C01818=1135.613,-74.660,-46.025,178.888,6.133,149.434
C01819=1135.619,-74.910,-46.015,178.885,6.132,149.434
C01820=1135.623,-75.160,-46.005,178.883,6.132,149.434
C01821=1135.629,-75.409,-45.995,178.881,6.131,149.435
C01822=1135.634,-75.659,-45.985,178.879,6.131,149.435
C01823=1135.639,-75.908,-45.975,178.877,6.130,149.436
C01824=1135.645,-76.158,-45.966,178.875,6.130,149.437
C01825=1135.650,-76.409,-45.955,178.872,6.129,149.437
C01826=1135.656,-76.679,-45.944,178.870,6.128,149.438
C01827=1135.662,-76.951,-45.934,178.867,6.128,149.438
C01828=1135.667,-77.223,-45.923,178.866,6.128,149.439
C01829=1135.674,-77.494,-45.912,178.864,6.127,149.439
C01830=1135.678,-77.744,-45.902,178.861,6.127,149.440
C01831=1135.684,-77.994,-45.892,178.859,6.126,149.440
C01832=1135.690,-78.244,-45.883,178.857,6.125,149.441
C01833=1135.695,-78.493,-45.873,178.855,6.125,149.441
C01834=1135.700,-78.743,-45.863,178.853,6.124,149.442
C01835=1135.706,-78.993,-45.853,178.851,6.124,149.442
C01836=1135.710,-79.243,-45.843,178.848,6.123,149.443
C01837=1135.716,-79.492,-45.833,178.846,6.123,149.444
C01838=1135.721,-79.742,-45.824,178.844,6.123,149.444
C01839=1135.727,-79.992,-45.814,178.842,6.122,149.445
C01840=1135.732,-80.241,-45.804,178.840,6.121,149.445
C01841=1135.738,-80.491,-45.795,178.838,6.121,149.446
C01842=1135.743,-80.741,-45.784,178.836,6.121,149.446
C01843=1135.747,-80.991,-45.775,178.833,6.120,149.447
C01844=1135.753,-81.241,-45.765,178.831,6.119,149.447
C01845=1135.759,-81.490,-45.755,178.830,6.119,149.448
C01846=1135.764,-81.739,-45.745,178.827,6.118,149.448
C01847=1135.770,-81.990,-45.736,178.825,6.118,149.449
C01848=1135.775,-82.239,-45.726,178.822,6.117,149.449
C01849=1135.780,-82.490,-45.716,178.821,6.117,149.450
C01850=1135.785,-82.739,-45.706,178.819,6.117,149.450
C01851=1135.790,-82.988,-45.697,178.817,6.116,149.451
C01852=1135.796,-83.239,-45.687,178.815,6.116,149.451
C01853=1135.801,-83.488,-45.677,178.812,6.116,149.452
C01854=1135.807,-83.738,-45.668,178.810,6.115,149.453
C01855=1135.812,-83.987,-45.658,178.808,6.114,149.453
C01856=1135.818,-84.237,-45.649,178.806,6.114,149.453
C01857=1135.822,-84.487,-45.639,178.804,6.113,149.454
C01858=1135.828,-84.738,-45.629,178.802,6.113,149.454
C01859=1135.833,-84.987,-45.620,178.799,6.112,149.455
C01860=1135.839,-85.237,-45.610,178.798,6.112,149.456
C01861=1135.843,-85.486,-45.601,178.795,6.111,149.456
C01862=1135.849,-85.736,-45.591,178.793,6.111,149.457
C01863=1135.854,-85.986,-45.582,178.792,6.111,149.457
C01864=1135.860,-86.236,-45.572,178.789,6.110,149.458
C01865=1135.865,-86.485,-45.562,178.787,6.109,149.458
C01866=1135.871,-86.735,-45.553,178.785,6.109,149.459
C01867=1135.876,-86.984,-45.543,178.783,6.109,149.459
C01868=1135.882,-87.235,-45.534,178.781,6.108,149.460
C01869=1135.886,-87.484,-45.524,178.779,6.107,149.460
C01870=1135.892,-87.735,-45.514,178.777,6.107,149.461
C01871=1135.897,-87.984,-45.505,178.775,6.107,149.461
C01872=1135.903,-88.234,-45.495,178.773,6.106,149.462
C01873=1135.908,-88.484,-45.486,178.771,6.106,149.462
C01874=1135.913,-88.733,-45.477,178.768,6.106,149.463
C01875=1135.919,-88.983,-45.467,178.766,6.105,149.463
C01876=1135.923,-89.232,-45.458,178.764,6.104,149.464
C01877=1135.929,-89.483,-45.448,178.762,6.104,149.464
C01878=1135.934,-89.733,-45.439,178.760,6.103,149.465
C01879=1135.940,-89.982,-45.429,178.758,6.103,149.465
C01880=1135.945,-90.232,-45.420,178.756,6.103,149.466
C01881=1135.950,-90.481,-45.411,178.754,6.102,149.466
C01882=1135.956,-90.731,-45.401,178.751,6.102,149.467
C01883=1135.961,-90.981,-45.392,178.750,6.102,149.467
C01884=1135.967,-91.231,-45.382,178.748,6.101,149.468
C01885=1135.972,-91.481,-45.373,178.745,6.100,149.468
C01886=1135.977,-91.730,-45.364,178.744,6.100,149.469
C01887=1135.983,-91.980,-45.354,178.742,6.099,149.469
C01888=1135.988,-92.230,-45.345,178.739,6.099,149.470
C01889=1135.994,-92.480,-45.336,178.737,6.098,149.471
C01890=1135.999,-92.729,-45.326,178.735,6.098,149.471
C01891=1136.004,-92.979,-45.317,178.733,6.098,149.472
C01892=1136.010,-93.229,-45.308,178.731,6.097,149.472
C01893=1136.015,-93.478,-45.298,178.729,6.097,149.473
C01894=1136.020,-93.728,-45.289,178.727,6.096,149.473
C01895=1136.026,-93.978,-45.280,178.725,6.095,149.474
C01896=1136.031,-94.228,-45.271,178.723,6.096,149.474
C01897=1136.036,-94.478,-45.261,178.721,6.095,149.475
C01898=1136.042,-94.728,-45.252,178.718,6.094,149.475
C01899=1136.047,-94.978,-45.243,178.717,6.094,149.476
C01900=1136.052,-95.227,-45.234,178.715,6.094,149.476
C01901=1136.058,-95.477,-45.224,178.712,6.093,149.477
C01902=1136.063,-95.727,-45.215,178.711,6.093,149.477
C01903=1136.068,-95.977,-45.206,178.709,6.092,149.478
C01904=1136.074,-96.227,-45.196,178.706,6.091,149.478
C01905=1136.079,-96.477,-45.187,178.704,6.092,149.479
C01906=1136.084,-96.725,-45.178,178.702,6.091,149.479
C01907=1136.090,-96.975,-45.169,178.700,6.090,149.480
C01908=1136.095,-97.225,-45.160,178.698,6.090,149.480
C01909=1136.101,-97.475,-45.151,178.696,6.090,149.481
C01910=1136.106,-97.725,-45.142,178.694,6.089,149.481
C01911=1136.111,-97.974,-45.132,178.692,6.089,149.482
C01912=1136.117,-98.224,-45.123,178.690,6.088,149.482
C01913=1136.122,-98.474,-45.114,178.689,6.088,149.483
C01914=1136.127,-98.724,-45.105,178.686,6.087,149.483
C01915=1136.133,-98.974,-45.096,178.684,6.087,149.484
C01916=1136.138,-99.224,-45.087,178.682,6.087,149.484
C01917=1136.143,-99.474,-45.078,178.680,6.086,149.485
C01918=1136.149,-99.722,-45.068,178.678,6.086,149.485
C01919=1136.154,-99.973,-45.059,178.676,6.086,149.486
C01920=1136.160,-100.222,-45.050,178.674,6.085,149.486
C01921=1136.165,-100.472,-45.041,178.672,6.084,149.487
C01922=1136.170,-100.722,-45.032,178.670,6.084,149.487
C01923=1136.175,-100.972,-45.023,178.668,6.083,149.488
C01924=1136.181,-101.222,-45.014,178.666,6.083,149.488
C01925=1136.186,-101.472,-45.005,178.664,6.083,149.489
C01926=1136.191,-101.722,-44.996,178.662,6.082,149.489
C01927=1136.197,-101.971,-44.988,178.660,6.082,149.490
C01928=1136.202,-102.221,-44.979,178.658,6.082,149.490
C01929=1136.208,-102.471,-44.969,178.655,6.081,149.491
C01930=1136.214,-102.743,-44.959,178.654,6.081,149.491
C01931=1136.220,-103.015,-44.949,178.652,6.080,149.492
C01932=1136.225,-103.287,-44.939,178.649,6.080,149.493
C01933=1136.231,-103.560,-44.930,178.647,6.079,149.493
C01934=1136.237,-103.809,-44.921,178.645,6.079,149.494
C01935=1136.242,-104.059,-44.912,178.643,6.078,149.494
C01936=1136.247,-104.309,-44.903,178.641,6.078,149.495
C01937=1136.252,-104.559,-44.894,178.639,6.078,149.495
C01938=1136.258,-104.809,-44.885,178.637,6.077,149.496
C01939=1136.263,-105.059,-44.876,178.635,6.076,149.496
C01940=1136.269,-105.308,-44.868,178.633,6.076,149.497
C01941=1136.274,-105.558,-44.859,178.631,6.075,149.497
C01942=1136.279,-105.807,-44.850,178.629,6.075,149.497
C01943=1136.284,-106.057,-44.841,178.627,6.075,149.498
C01944=1136.290,-106.307,-44.832,178.625,6.074,149.498
C01945=1136.295,-106.557,-44.823,178.623,6.074,149.499
C01946=1136.301,-106.806,-44.815,178.621,6.074,149.500
C01947=1136.306,-107.056,-44.805,178.619,6.074,149.500
C01948=1136.312,-107.306,-44.796,178.617,6.073,149.501
C01949=1136.317,-107.557,-44.788,178.615,6.072,149.501
C01950=1136.322,-107.807,-44.779,178.613,6.072,149.502
C01951=1136.328,-108.056,-44.771,178.611,6.071,149.502
C01952=1136.333,-108.306,-44.762,178.609,6.072,149.503
C01953=1136.338,-108.555,-44.753,178.607,6.071,149.503
C01954=1136.343,-108.805,-44.744,178.605,6.070,149.504
C01955=1136.349,-109.055,-44.735,178.603,6.070,149.504
C01956=1136.354,-109.304,-44.726,178.601,6.069,149.505
C01957=1136.360,-109.554,-44.717,178.600,6.069,149.505
C01958=1136.365,-109.805,-44.709,178.597,6.069,149.505
C01959=1136.370,-110.054,-44.700,178.595,6.068,149.506
C01960=1136.376,-110.304,-44.692,178.594,6.068,149.506
C01961=1136.381,-110.553,-44.683,178.591,6.067,149.507
C01962=1136.386,-110.803,-44.674,178.590,6.067,149.507
C01963=1136.391,-111.053,-44.665,178.588,6.066,149.508
C01964=1136.398,-111.303,-44.657,178.585,6.066,149.508
C01965=1136.403,-111.553,-44.648,178.584,6.066,149.509
C01966=1136.408,-111.803,-44.640,178.582,6.065,149.509
C01967=1136.413,-112.052,-44.631,178.580,6.065,149.510
C01968=1136.419,-112.302,-44.622,178.578,6.064,149.510
C01969=1136.424,-112.551,-44.613,178.576,6.065,149.511
C01970=1136.429,-112.802,-44.605,178.574,6.064,149.512
C01971=1136.435,-113.052,-44.596,178.571,6.063,149.512
C01972=1136.440,-113.301,-44.588,178.570,6.063,149.513
C01973=1136.446,-113.551,-44.579,178.568,6.063,149.513
C01974=1136.451,-113.801,-44.571,178.566,6.063,149.514
C01975=1136.457,-114.050,-44.562,178.564,6.062,149.514
C01976=1136.462,-114.300,-44.553,178.562,6.062,149.514
C01977=1136.467,-114.550,-44.544,178.560,6.061,149.515
C01978=1136.473,-114.801,-44.536,178.558,6.060,149.515
C01979=1136.478,-115.050,-44.528,178.556,6.060,149.516
C01980=1136.484,-115.300,-44.519,178.554,6.060,149.516
C01981=1136.489,-115.549,-44.510,178.552,6.060,149.517
C01982=1136.495,-115.799,-44.502,178.550,6.059,149.517
C01983=1136.500,-116.049,-44.493,178.549,6.059,149.518
C01984=1136.505,-116.299,-44.484,178.546,6.058,149.518
C01985=1136.511,-116.549,-44.476,178.544,6.058,149.519
C01986=1136.516,-116.798,-44.467,178.543,6.058,149.519
C01987=1136.522,-117.048,-44.458,178.540,6.057,149.520
C01988=1136.528,-117.298,-44.451,178.539,6.057,149.520
C01989=1136.532,-117.548,-44.442,178.537,6.056,149.521
C01990=1136.537,-117.798,-44.433,178.535,6.056,149.521
C01991=1136.543,-118.047,-44.426,178.533,6.055,149.522
C01992=1136.548,-118.297,-44.417,178.531,6.056,149.522
C01993=1136.554,-118.547,-44.408,178.529,6.055,149.523
C01994=1136.560,-118.797,-44.400,178.527,6.054,149.523
C01995=1136.565,-119.047,-44.391,178.525,6.054,149.524
C01996=1136.570,-119.297,-44.383,178.523,6.053,149.524
C01997=1136.575,-119.546,-44.375,178.521,6.053,149.525
C01998=1136.581,-119.796,-44.366,178.519,6.053,149.525
C01999=1136.586,-120.046,-44.358,178.518,6.053,149.526
C02000=1136.592,-120.295,-44.349,178.515,6.052,149.526
C02001=1136.597,-120.545,-44.341,178.514,6.052,149.527
C02002=1136.602,-120.796,-44.332,178.512,6.051,149.527
C02003=1136.608,-121.045,-44.324,178.510,6.051,149.528
C02004=1136.613,-121.295,-44.316,178.508,6.051,149.528
C02005=1136.619,-121.544,-44.308,178.506,6.050,149.529
C02006=1136.624,-121.795,-44.300,178.505,6.049,149.529
C02007=1136.629,-122.044,-44.291,178.502,6.049,149.529
C02008=1136.635,-122.294,-44.282,178.501,6.049,149.530
C02009=1136.640,-122.544,-44.274,178.499,6.048,149.530
C02010=1136.645,-122.794,-44.266,178.497,6.048,149.531
C02011=1136.651,-123.043,-44.258,178.495,6.047,149.531
C02012=1136.656,-123.293,-44.249,178.493,6.047,149.532
C02013=1136.662,-123.543,-44.241,178.491,6.047,149.532
C02014=1136.667,-123.793,-44.233,178.489,6.047,149.533
C02015=1136.672,-124.043,-44.225,178.487,6.046,149.533
C02016=1136.678,-124.292,-44.216,178.486,6.046,149.534
C02017=1136.683,-124.543,-44.208,178.483,6.045,149.534
C02018=1136.689,-124.792,-44.199,178.482,6.045,149.535
C02019=1136.694,-125.042,-44.192,178.480,6.045,149.535
C02020=1136.700,-125.291,-44.183,178.478,6.045,149.536
C02021=1136.705,-125.542,-44.175,178.476,6.044,149.536
C02022=1136.710,-125.791,-44.166,178.474,6.043,149.537
C02023=1136.716,-126.041,-44.159,178.472,6.043,149.537
C02024=1136.721,-126.291,-44.151,178.470,6.042,149.538
C02025=1136.727,-126.541,-44.142,178.468,6.042,149.538
C02026=1136.732,-126.791,-44.134,178.466,6.042,149.539
C02027=1136.737,-127.040,-44.126,178.464,6.042,149.539
C02028=1136.743,-127.290,-44.118,178.462,6.041,149.540
C02029=1136.748,-127.540,-44.109,178.461,6.041,149.540
C02030=1136.753,-127.790,-44.102,178.459,6.040,149.540
C02031=1136.759,-128.040,-44.094,178.457,6.040,149.541
C02032=1136.765,-128.289,-44.085,178.455,6.039,149.541
C02033=1136.770,-128.540,-44.077,178.454,6.039,149.542
C02034=1136.349,-128.551,-44.121,178.450,6.043,149.544
C02035=1136.344,-128.300,-44.129,178.452,6.043,149.543
C02036=1136.337,-128.051,-44.137,178.453,6.043,149.543
C02037=1136.333,-127.801,-44.145,178.456,6.044,149.542
C02038=1136.327,-127.551,-44.153,178.457,6.044,149.542
C02039=1136.322,-127.301,-44.162,178.459,6.045,149.541
C02040=1136.316,-127.052,-44.169,178.461,6.045,149.541
C02041=1136.311,-126.802,-44.178,178.463,6.045,149.540
C02042=1136.306,-126.552,-44.186,178.465,6.045,149.540
C02043=1136.300,-126.302,-44.194,178.467,6.046,149.539
C02044=1136.295,-126.052,-44.202,178.469,6.046,149.539
C02045=1136.289,-125.803,-44.210,178.470,6.047,149.539
C02046=1136.284,-125.553,-44.219,178.473,6.048,149.538
C02047=1136.278,-125.303,-44.227,178.474,6.048,149.538
C02048=1136.274,-125.053,-44.235,178.476,6.049,149.537
C02049=1136.268,-124.803,-44.243,178.478,6.049,149.537
C02050=1136.262,-124.554,-44.252,178.480,6.049,149.536
C02051=1136.257,-124.303,-44.260,178.482,6.049,149.536
C02052=1136.252,-124.054,-44.268,178.484,6.050,149.535
C02053=1136.246,-123.804,-44.276,178.486,6.050,149.535
C02054=1136.241,-123.554,-44.285,178.488,6.051,149.534
C02055=1136.235,-123.304,-44.293,178.489,6.051,149.534
C02056=1136.230,-123.055,-44.302,178.492,6.051,149.533
C02057=1136.225,-122.805,-44.309,178.493,6.051,149.533
C02058=1136.219,-122.555,-44.318,178.495,6.052,149.532
C02059=1136.214,-122.305,-44.326,178.497,6.052,149.532
C02060=1136.208,-122.056,-44.335,178.499,6.053,149.531
C02061=1136.203,-121.805,-44.343,178.501,6.053,149.531
C02062=1136.198,-121.556,-44.351,178.503,6.053,149.530
C02063=1136.193,-121.306,-44.360,178.505,6.054,149.530
C02064=1136.187,-121.056,-44.368,178.507,6.054,149.529
C02065=1136.181,-120.807,-44.376,178.509,6.055,149.529
C02066=1136.176,-120.556,-44.385,178.511,6.055,149.528
C02067=1136.171,-120.306,-44.394,178.513,6.056,149.528
C02068=1136.165,-120.057,-44.401,178.514,6.056,149.527
C02069=1136.160,-119.807,-44.410,178.517,6.056,149.527
C02070=1136.155,-119.557,-44.419,178.518,6.056,149.526
C02071=1136.149,-119.308,-44.426,178.520,6.057,149.526
C02072=1136.144,-119.058,-44.435,178.521,6.057,149.526
C02073=1136.138,-118.809,-44.444,178.524,6.058,149.525
C02074=1136.133,-118.558,-44.452,178.526,6.059,149.525
C02075=1136.128,-118.309,-44.460,178.527,6.059,149.524
C02076=1136.122,-118.059,-44.468,178.530,6.060,149.524
C02077=1136.117,-117.809,-44.477,178.531,6.059,149.523
C02078=1136.112,-117.559,-44.486,178.533,6.060,149.523
C02079=1136.106,-117.309,-44.494,178.535,6.060,149.522
C02080=1136.100,-117.059,-44.503,178.537,6.061,149.522
C02081=1136.095,-116.810,-44.512,178.539,6.061,149.521
C02082=1136.089,-116.560,-44.519,178.541,6.062,149.521
C02083=1136.084,-116.310,-44.528,178.543,6.062,149.520
C02084=1136.079,-116.060,-44.537,178.545,6.062,149.520
C02085=1136.074,-115.810,-44.546,178.547,6.063,149.519
C02086=1136.068,-115.561,-44.554,178.549,6.063,149.519
C02087=1136.063,-115.311,-44.562,178.551,6.064,149.518
C02088=1136.058,-115.061,-44.571,178.552,6.064,149.518
C02089=1136.052,-114.811,-44.579,178.555,6.064,149.517
C02090=1136.047,-114.562,-44.588,178.556,6.064,149.517
C02091=1136.042,-114.312,-44.597,178.558,6.065,149.516
C02092=1136.036,-114.063,-44.605,178.561,6.066,149.516
C02093=1136.030,-113.812,-44.613,178.562,6.066,149.515
C02094=1136.025,-113.562,-44.622,178.564,6.067,149.515
C02095=1136.020,-113.312,-44.631,178.566,6.066,149.514
C02096=1136.014,-113.063,-44.640,178.569,6.067,149.514
C02097=1136.009,-112.813,-44.648,178.571,6.068,149.513
C02098=1136.004,-112.563,-44.657,178.572,6.068,149.513
C02099=1135.998,-112.314,-44.665,178.575,6.068,149.512
C02100=1135.993,-112.064,-44.674,178.576,6.068,149.512
C02101=1135.988,-111.814,-44.683,178.578,6.069,149.511
C02102=1135.982,-111.564,-44.691,178.580,6.069,149.511
C02103=1135.976,-111.314,-44.700,178.582,6.070,149.510
C02104=1135.971,-111.065,-44.709,178.584,6.071,149.510
C02105=1135.966,-110.815,-44.718,178.586,6.070,149.509
C02106=1135.961,-110.565,-44.727,178.588,6.071,149.509
C02107=1135.955,-110.315,-44.734,178.590,6.071,149.508
C02108=1135.950,-110.065,-44.743,178.592,6.072,149.508
C02109=1135.944,-109.815,-44.752,178.594,6.073,149.507
C02110=1135.939,-109.566,-44.761,178.596,6.073,149.507
C02111=1135.933,-109.316,-44.770,178.598,6.073,149.506
C02112=1135.928,-109.067,-44.778,178.600,6.073,149.506
C02113=1135.923,-108.817,-44.787,178.602,6.074,149.505
C02114=1135.918,-108.567,-44.796,178.604,6.075,149.505
C02115=1135.912,-108.316,-44.805,178.606,6.075,149.504
C02116=1135.906,-108.067,-44.814,178.608,6.076,149.504
C02117=1135.901,-107.817,-44.822,178.609,6.075,149.503
C02118=1135.896,-107.567,-44.831,178.612,6.076,149.503
C02119=1135.891,-107.317,-44.840,178.614,6.077,149.502
C02120=1135.885,-107.067,-44.849,178.615,6.077,149.502
C02121=1135.880,-106.818,-44.858,178.618,6.078,149.501
C02122=1135.874,-106.568,-44.867,178.619,6.078,149.501
C02123=1135.869,-106.319,-44.875,178.621,6.078,149.500
C02124=1135.864,-106.069,-44.884,178.624,6.079,149.500
C02125=1135.859,-105.819,-44.893,178.626,6.079,149.499
C02126=1135.853,-105.570,-44.902,178.628,6.079,149.499
C02127=1135.847,-105.320,-44.911,178.629,6.079,149.498
C02128=1135.842,-105.070,-44.920,178.632,6.080,149.498
C02129=1135.837,-104.820,-44.929,178.634,6.081,149.497
C02130=1135.832,-104.570,-44.938,178.635,6.081,149.497
C02131=1135.827,-104.320,-44.947,178.638,6.082,149.496
C02132=1135.821,-104.071,-44.955,178.640,6.082,149.496
C02133=1135.816,-103.821,-44.964,178.641,6.082,149.495
C02134=1135.810,-103.571,-44.974,178.644,6.083,149.495
C02135=1135.804,-103.298,-44.983,178.646,6.084,149.494
C02136=1135.798,-103.026,-44.993,178.648,6.083,149.494
C02137=1135.793,-102.754,-45.003,178.650,6.084,149.493
C02138=1135.787,-102.481,-45.013,178.652,6.085,149.493
C02139=1135.781,-102.232,-45.021,178.654,6.085,149.492
C02140=1135.776,-101.982,-45.030,178.656,6.086,149.492
C02141=1135.771,-101.733,-45.039,178.658,6.086,149.491
C02142=1135.765,-101.482,-45.048,178.660,6.086,149.491
C02143=1135.760,-101.233,-45.057,178.663,6.087,149.490
C02144=1135.754,-100.983,-45.066,178.665,6.087,149.490
C02145=1135.750,-100.734,-45.076,178.666,6.087,149.489
C02146=1135.744,-100.484,-45.085,178.669,6.088,149.489
C02147=1135.738,-100.234,-45.094,178.671,6.089,149.488
C02148=1135.733,-99.984,-45.103,178.672,6.089,149.488
C02149=1135.728,-99.735,-45.112,178.674,6.090,149.487
C02150=1135.722,-99.485,-45.121,178.677,6.090,149.487
C02151=1135.717,-99.234,-45.130,178.678,6.090,149.486
C02152=1135.711,-98.985,-45.139,178.680,6.091,149.486
C02153=1135.706,-98.735,-45.148,178.682,6.091,149.485
C02154=1135.701,-98.486,-45.157,178.684,6.092,149.485
C02155=1135.695,-98.235,-45.167,178.687,6.092,149.484
C02156=1135.690,-97.986,-45.176,178.689,6.092,149.484
C02157=1135.685,-97.736,-45.184,178.691,6.093,149.483
C02158=1135.679,-97.487,-45.193,178.693,6.094,149.483
C02159=1135.673,-97.236,-45.203,178.695,6.094,149.482
C02160=1135.669,-96.987,-45.212,178.697,6.094,149.482
C02161=1135.663,-96.737,-45.221,178.699,6.095,149.481
C02162=1135.658,-96.487,-45.230,178.701,6.095,149.481
C02163=1135.652,-96.237,-45.240,178.703,6.096,149.480
C02164=1135.647,-95.987,-45.249,178.705,6.096,149.480
C02165=1135.642,-95.738,-45.258,178.707,6.096,149.479
C02166=1135.636,-95.488,-45.268,178.709,6.097,149.478
C02167=1135.631,-95.238,-45.277,178.711,6.098,149.478
C02168=1135.626,-94.988,-45.285,178.713,6.098,149.477
C02169=1135.621,-94.739,-45.296,178.715,6.098,149.477
C02170=1135.615,-94.489,-45.305,178.717,6.099,149.477
C02171=1135.610,-94.239,-45.313,178.719,6.099,149.476
C02172=1135.604,-93.989,-45.323,178.721,6.100,149.476
C02173=1135.599,-93.740,-45.333,178.723,6.100,149.475
C02174=1135.594,-93.490,-45.341,178.725,6.100,149.474
C02175=1135.588,-93.240,-45.351,178.728,6.101,149.474
C02176=1135.583,-92.990,-45.360,178.730,6.102,149.473
C02177=1135.578,-92.741,-45.369,178.731,6.102,149.473
C02178=1135.572,-92.490,-45.379,178.734,6.102,149.472
C02179=1135.567,-92.241,-45.388,178.736,6.103,149.472
C02180=1135.562,-91.991,-45.398,178.737,6.103,149.471
C02181=1135.556,-91.741,-45.407,178.740,6.104,149.471
C02182=1135.551,-91.491,-45.416,178.742,6.104,149.470
C02183=1135.546,-91.242,-45.426,178.744,6.104,149.470
C02184=1135.541,-90.992,-45.435,178.746,6.105,149.469
C02185=1135.535,-90.742,-45.444,178.748,6.106,149.469
C02186=1135.530,-90.493,-45.454,178.750,6.106,149.468
C02187=1135.525,-90.243,-45.463,178.752,6.106,149.468
C02188=1135.519,-89.993,-45.472,178.754,6.107,149.467
C02189=1135.514,-89.743,-45.482,178.756,6.108,149.467
C02190=1135.508,-89.493,-45.492,178.758,6.107,149.466
C02191=1135.503,-89.244,-45.501,178.761,6.108,149.466
C02192=1135.498,-88.994,-45.510,178.763,6.109,149.465
C02193=1135.492,-88.744,-45.520,178.764,6.109,149.465
C02194=1135.487,-88.495,-45.529,178.767,6.110,149.464
C02195=1135.481,-88.244,-45.539,178.769,6.110,149.464
C02196=1135.476,-87.995,-45.548,178.771,6.111,149.463
C02197=1135.470,-87.745,-45.558,178.773,6.111,149.463
C02198=1135.466,-87.496,-45.567,178.775,6.111,149.462
C02199=1135.460,-87.246,-45.576,178.778,6.112,149.462
C02200=1135.455,-86.996,-45.586,178.779,6.112,149.461
C02201=1135.450,-86.747,-45.595,178.781,6.113,149.461
C02202=1135.444,-86.496,-45.605,178.784,6.114,149.460
C02203=1135.439,-86.247,-45.615,178.785,6.114,149.460
C02204=1135.433,-85.997,-45.624,178.787,6.114,149.459
C02205=1135.429,-85.747,-45.634,178.790,6.115,149.458
C02206=1135.423,-85.497,-45.643,178.792,6.115,149.458
C02207=1135.418,-85.248,-45.653,178.794,6.115,149.457
C02208=1135.412,-84.998,-45.663,178.796,6.116,149.457
C02209=1135.407,-84.748,-45.672,178.798,6.117,149.456
C02210=1135.401,-84.498,-45.682,178.800,6.118,149.456
C02211=1135.396,-84.249,-45.691,178.802,6.117,149.455
C02212=1135.391,-83.999,-45.701,178.805,6.118,149.455
C02213=1135.386,-83.750,-45.710,178.807,6.119,149.454
C02214=1135.380,-83.500,-45.721,178.808,6.119,149.454
C02215=1135.375,-83.249,-45.730,178.811,6.120,149.453
C02216=1135.370,-83.000,-45.740,178.813,6.120,149.453
C02217=1135.364,-82.750,-45.750,178.815,6.121,149.452
C02218=1135.359,-82.501,-45.759,178.817,6.121,149.452
C02219=1135.353,-82.250,-45.769,178.819,6.121,149.451
C02220=1135.348,-82.001,-45.778,178.821,6.122,149.451
C02221=1135.343,-81.752,-45.789,178.824,6.123,149.450
C02222=1135.337,-81.501,-45.798,178.825,6.123,149.450
C02223=1135.333,-81.251,-45.808,178.827,6.124,149.449
C02224=1135.327,-81.001,-45.817,178.830,6.124,149.449
C02225=1135.322,-80.752,-45.827,178.832,6.125,149.448
C02226=1135.316,-80.503,-45.837,178.834,6.125,149.448
C02227=1135.311,-80.253,-45.846,178.836,6.125,149.447
C02228=1135.306,-80.003,-45.856,178.838,6.126,149.447
C02229=1135.301,-79.753,-45.867,178.841,6.127,149.446
C02230=1135.295,-79.503,-45.876,178.843,6.127,149.445
C02231=1135.290,-79.254,-45.886,178.845,6.127,149.445
C02232=1135.284,-79.004,-45.896,178.847,6.128,149.444
C02233=1135.279,-78.754,-45.905,178.849,6.129,149.444
C02234=1135.273,-78.505,-45.915,178.851,6.129,149.444
C02235=1135.268,-78.254,-45.926,178.853,6.129,149.443
C02236=1135.263,-78.004,-45.935,178.856,6.130,149.442
C02237=1135.258,-77.755,-45.945,178.858,6.131,149.442
C02238=1135.252,-77.505,-45.955,178.859,6.131,149.441
C02239=1135.247,-77.233,-45.966,178.862,6.131,149.441
C02240=1135.241,-76.963,-45.976,178.864,6.132,149.440
C02241=1135.235,-76.691,-45.987,178.866,6.133,149.440
C02242=1135.229,-76.419,-45.998,178.869,6.133,149.439
C02243=1135.224,-76.170,-46.008,178.871,6.134,149.438
C02244=1135.218,-75.920,-46.018,178.874,6.134,149.438
C02245=1135.213,-75.670,-46.027,178.875,6.134,149.438
C02246=1135.208,-75.420,-46.038,178.877,6.135,149.437
C02247=1135.202,-75.171,-46.048,178.880,6.136,149.436
C02248=1135.197,-74.921,-46.058,178.882,6.136,149.436
C02249=1135.192,-74.671,-46.067,178.884,6.136,149.435
C02250=1135.187,-74.421,-46.078,178.886,6.137,149.435
C02251=1135.181,-74.171,-46.088,178.888,6.138,149.434
C02252=1135.176,-73.922,-46.097,178.890,6.139,149.434
C02253=1135.171,-73.673,-46.108,178.892,6.138,149.433
C02254=1135.166,-73.422,-46.118,178.895,6.139,149.433
C02255=1135.160,-73.172,-46.128,178.897,6.140,149.432
C02256=1135.154,-72.923,-46.138,178.899,6.140,149.432
C02257=1135.149,-72.673,-46.148,178.901,6.141,149.431
C02258=1135.144,-72.423,-46.158,178.903,6.141,149.431
C02259=1135.139,-72.174,-46.168,178.905,6.142,149.430
C02260=1135.133,-71.924,-46.179,178.908,6.142,149.430
C02261=1135.128,-71.675,-46.188,178.910,6.143,149.429
C02262=1135.123,-71.424,-46.198,178.912,6.144,149.429
C02263=1135.117,-71.175,-46.208,178.914,6.143,149.428
C02264=1135.112,-70.925,-46.218,178.916,6.144,149.427
C02265=1135.106,-70.675,-46.229,178.918,6.145,149.427
C02266=1135.102,-70.426,-46.239,178.921,6.146,149.426
C02267=1135.096,-70.176,-46.249,178.923,6.146,149.426
C02268=1135.091,-69.926,-46.259,178.925,6.146,149.425
C02269=1135.086,-69.676,-46.270,178.927,6.147,149.425
C02270=1135.080,-69.427,-46.280,178.929,6.148,149.424
C02271=1135.074,-69.177,-46.290,178.932,6.148,149.424
C02272=1135.070,-68.927,-46.300,178.934,6.149,149.423
C02273=1135.065,-68.678,-46.310,178.936,6.149,149.423
C02274=1135.059,-68.428,-46.320,178.938,6.149,149.422
C02275=1135.053,-68.179,-46.331,178.940,6.150,149.422
C02276=1135.048,-67.928,-46.341,178.942,6.151,149.421
C02277=1135.043,-67.679,-46.351,178.945,6.151,149.420
C02278=1135.037,-67.429,-46.362,178.947,6.151,149.420
C02279=1135.033,-67.179,-46.372,178.949,6.152,149.420
C02280=1135.027,-66.930,-46.382,178.951,6.153,149.419
C02281=1135.022,-66.680,-46.392,178.953,6.154,149.419
C02282=1135.017,-66.430,-46.403,178.956,6.154,149.418
C02283=1135.011,-66.180,-46.413,178.958,6.155,149.417
C02284=1135.006,-65.930,-46.423,178.960,6.155,149.417
C02285=1135.000,-65.681,-46.434,178.962,6.155,149.416
C02286=1134.995,-65.431,-46.444,178.965,6.156,149.416
C02287=1134.990,-65.181,-46.454,178.967,6.157,149.415
C02288=1134.984,-64.931,-46.465,178.969,6.157,149.415
C02289=1134.979,-64.682,-46.474,178.971,6.158,149.414
C02290=1134.974,-64.432,-46.485,178.973,6.158,149.414
C02291=1134.969,-64.182,-46.495,178.975,6.158,149.413
C02292=1134.963,-63.933,-46.505,178.978,6.159,149.413
C02293=1134.959,-63.683,-46.516,178.980,6.160,149.412
C02294=1134.953,-63.434,-46.527,178.982,6.161,149.412
C02295=1134.948,-63.183,-46.537,178.985,6.161,149.411
C02296=1134.942,-62.934,-46.547,178.986,6.161,149.410
C02297=1134.937,-62.684,-46.558,178.988,6.162,149.410
C02298=1134.932,-62.434,-46.568,178.991,6.163,149.409
C02299=1134.926,-62.184,-46.578,178.993,6.163,149.409
C02300=1134.921,-61.935,-46.590,178.995,6.164,149.408
C02301=1134.916,-61.685,-46.600,178.998,6.165,149.408
C02302=1134.911,-61.435,-46.611,179.000,6.165,149.407
C02303=1134.905,-61.185,-46.621,179.002,6.165,149.407
C02304=1134.900,-60.936,-46.631,179.004,6.166,149.406
C02305=1134.895,-60.686,-46.642,179.006,6.166,149.406
C02306=1134.889,-60.437,-46.652,179.008,6.167,149.405
C02307=1134.884,-60.186,-46.663,179.011,6.168,149.405
C02308=1134.879,-59.937,-46.673,179.013,6.168,149.404
C02309=1134.874,-59.687,-46.684,179.015,6.168,149.404
C02310=1134.869,-59.438,-46.695,179.017,6.169,149.403
C02311=1134.863,-59.188,-46.705,179.019,6.170,149.403
C02312=1134.858,-58.938,-46.716,179.022,6.170,149.402
C02313=1134.852,-58.688,-46.726,179.024,6.171,149.401
C02314=1134.848,-58.439,-46.737,179.026,6.172,149.401
C02315=1134.842,-58.189,-46.747,179.029,6.173,149.400
C02316=1134.837,-57.939,-46.758,179.031,6.173,149.400
C02317=1134.832,-57.690,-46.769,179.033,6.173,149.399
C02318=1134.827,-57.440,-46.779,179.035,6.174,149.399
C02319=1134.821,-57.190,-46.790,179.037,6.174,149.398
C02320=1134.815,-56.940,-46.801,179.040,6.175,149.398
C02321=1134.810,-56.691,-46.812,179.042,6.176,149.397
C02322=1134.805,-56.441,-46.822,179.044,6.176,149.397
C02323=1134.800,-56.191,-46.832,179.046,6.177,149.396
C02324=1134.795,-55.941,-46.844,179.049,6.178,149.395
C02325=1134.789,-55.692,-46.854,179.051,6.178,149.395
C02326=1134.785,-55.442,-46.865,179.053,6.178,149.394
C02327=1134.779,-55.193,-46.875,179.055,6.179,149.394
C02328=1134.774,-54.942,-46.886,179.058,6.179,149.393
C02329=1134.768,-54.693,-46.897,179.060,6.180,149.393
C02330=1134.763,-54.443,-46.908,179.062,6.181,149.392
C02331=1134.757,-54.193,-46.918,179.064,6.182,149.392
C02332=1134.753,-53.944,-46.930,179.067,6.182,149.391
C02333=1134.747,-53.694,-46.940,179.069,6.183,149.391
C02334=1134.742,-53.445,-46.951,179.071,6.183,149.390
C02335=1134.737,-53.194,-46.962,179.073,6.184,149.390
C02336=1134.731,-52.945,-46.973,179.076,6.184,149.389
C02337=1134.726,-52.695,-46.984,179.078,6.185,149.389
C02338=1134.721,-52.445,-46.994,179.080,6.186,149.388
C02339=1134.716,-52.196,-47.005,179.083,6.186,149.387
C02340=1134.710,-51.946,-47.015,179.085,6.187,149.387
C02341=1134.705,-51.696,-47.027,179.087,6.187,149.386
C02342=1134.699,-51.447,-47.038,179.089,6.188,149.386
C02343=1134.694,-51.176,-47.050,179.092,6.189,149.385
C02344=1134.689,-50.905,-47.061,179.094,6.189,149.385
C02345=1134.683,-50.635,-47.073,179.097,6.190,149.384
C02346=1134.677,-50.363,-47.085,179.099,6.191,149.384
C02347=1134.672,-50.114,-47.096,179.101,6.191,149.383
C02348=1134.666,-49.864,-47.106,179.104,6.192,149.382
C02349=1134.661,-49.614,-47.118,179.106,6.192,149.382
C02350=1134.656,-49.365,-47.129,179.108,6.193,149.381
C02351=1134.651,-49.115,-47.140,179.110,6.194,149.381
C02352=1134.645,-48.866,-47.151,179.113,6.194,149.380
C02353=1134.640,-48.615,-47.162,179.115,6.194,149.380
C02354=1134.635,-48.366,-47.173,179.117,6.195,149.379
C02355=1134.629,-48.116,-47.183,179.119,6.196,149.379
C02356=1134.625,-47.867,-47.195,179.122,6.196,149.378
C02357=1134.619,-47.617,-47.206,179.124,6.197,149.378
C02358=1134.614,-47.367,-47.217,179.126,6.198,149.377
C02359=1134.609,-47.118,-47.228,179.129,6.198,149.376
C02360=1134.603,-46.868,-47.239,179.131,6.199,149.376
C02361=1134.598,-46.618,-47.250,179.133,6.200,149.375
C02362=1134.593,-46.368,-47.261,179.135,6.201,149.375
C02363=1134.587,-46.119,-47.272,179.138,6.201,149.374
C02364=1134.582,-45.869,-47.283,179.140,6.202,149.374
C02365=1134.578,-45.619,-47.295,179.142,6.203,149.373
C02366=1134.571,-45.369,-47.306,179.145,6.203,149.373
C02367=1134.567,-45.120,-47.317,179.147,6.204,149.372
C02368=1134.562,-44.870,-47.328,179.149,6.204,149.372
C02369=1134.556,-44.620,-47.339,179.151,6.204,149.371
C02370=1134.551,-44.371,-47.350,179.154,6.205,149.370
C02371=1134.546,-44.121,-47.362,179.156,6.206,149.370
C02372=1134.540,-43.871,-47.372,179.158,6.206,149.370
C02373=1134.535,-43.622,-47.384,179.161,6.207,149.369
C02374=1134.530,-43.372,-47.396,179.163,6.208,149.368
C02375=1134.524,-43.123,-47.406,179.165,6.208,149.368
C02376=1134.519,-42.873,-47.417,179.167,6.209,149.367
C02377=1134.514,-42.623,-47.429,179.170,6.209,149.367
C02378=1134.509,-42.374,-47.440,179.172,6.210,149.366
C02379=1134.503,-42.124,-47.452,179.174,6.211,149.366
C02380=1134.498,-41.874,-47.462,179.177,6.211,149.365
C02381=1134.494,-41.624,-47.474,179.179,6.212,149.365
C02382=1134.488,-41.375,-47.485,179.181,6.213,149.364
C02383=1134.483,-41.125,-47.496,179.184,6.214,149.364
C02384=1134.477,-40.875,-47.508,179.186,6.214,149.363
C02385=1134.472,-40.626,-47.518,179.188,6.215,149.362
C02386=1134.466,-40.376,-47.530,179.191,6.216,149.362
C02387=1134.462,-40.126,-47.542,179.193,6.216,149.361
C02388=1134.456,-39.876,-47.554,179.195,6.217,149.361
C02389=1134.451,-39.627,-47.564,179.198,6.218,149.360
C02390=1134.445,-39.377,-47.576,179.200,6.218,149.360
C02391=1134.441,-39.127,-47.587,179.202,6.219,149.359
C02392=1134.434,-38.878,-47.598,179.205,6.220,149.359
C02393=1134.430,-38.628,-47.610,179.207,6.220,149.358
C02394=1134.424,-38.378,-47.622,179.210,6.221,149.357
C02395=1134.420,-38.129,-47.633,179.212,6.222,149.357
C02396=1134.414,-37.879,-47.645,179.214,6.222,149.357
C02397=1134.409,-37.630,-47.656,179.217,6.223,149.356
C02398=1134.404,-37.380,-47.668,179.219,6.224,149.355
C02399=1134.399,-37.129,-47.678,179.221,6.224,149.355
C02400=1134.393,-36.880,-47.690,179.223,6.225,149.354
C02401=1134.388,-36.631,-47.701,179.226,6.225,149.354
C02402=1134.382,-36.381,-47.713,179.228,6.226,149.353
C02403=1134.378,-36.131,-47.724,179.230,6.227,149.353
C02404=1134.372,-35.881,-47.736,179.233,6.227,149.352
C02405=1134.368,-35.631,-47.747,179.235,6.228,149.352
C02406=1134.362,-35.382,-47.759,179.237,6.229,149.351
C02407=1134.356,-35.132,-47.771,179.239,6.230,149.351
C02408=1134.351,-34.883,-47.782,179.242,6.230,149.350
C02409=1134.346,-34.633,-47.794,179.244,6.231,149.349
C02410=1134.341,-34.383,-47.805,179.246,6.232,149.349
C02411=1134.335,-34.134,-47.817,179.249,6.232,149.348
C02412=1134.330,-33.884,-47.829,179.251,6.233,149.348
C02413=1134.325,-33.634,-47.840,179.253,6.234,149.347
C02414=1134.320,-33.384,-47.852,179.256,6.234,149.347
C02415=1134.315,-33.135,-47.863,179.258,6.235,149.346
C02416=1134.310,-32.885,-47.875,179.260,6.236,149.346
C02417=1134.304,-32.636,-47.886,179.263,6.236,149.345
C02418=1134.299,-32.386,-47.898,179.265,6.237,149.344
C02419=1134.293,-32.136,-47.910,179.268,6.238,149.344
C02420=1134.288,-31.887,-47.922,179.270,6.238,149.344
C02421=1134.284,-31.637,-47.934,179.272,6.239,149.343
C02422=1134.278,-31.387,-47.945,179.275,6.240,149.342
C02423=1134.273,-31.138,-47.957,179.277,6.240,149.342
C02424=1134.267,-30.888,-47.968,179.279,6.241,149.341
C02425=1134.262,-30.638,-47.980,179.282,6.242,149.341
C02426=1134.257,-30.389,-47.991,179.284,6.242,149.340
C02427=1134.252,-30.139,-48.003,179.286,6.243,149.340
C02428=1134.247,-29.889,-48.016,179.289,6.243,149.339
C02429=1134.241,-29.640,-48.028,179.291,6.244,149.339
C02430=1134.237,-29.390,-48.039,179.293,6.245,149.338
C02431=1134.231,-29.140,-48.051,179.296,6.245,149.337
C02432=1134.226,-28.890,-48.063,179.298,6.246,149.337
C02433=1134.221,-28.641,-48.074,179.300,6.247,149.336
C02434=1134.215,-28.392,-48.086,179.303,6.248,149.336
C02435=1134.210,-28.142,-48.098,179.305,6.249,149.335
C02436=1134.205,-27.892,-48.110,179.308,6.250,149.335
C02437=1134.200,-27.642,-48.121,179.310,6.250,149.334
C02438=1134.195,-27.393,-48.134,179.313,6.251,149.334
C02439=1134.189,-27.143,-48.146,179.315,6.252,149.333
C02440=1134.184,-26.893,-48.158,179.317,6.252,149.332
C02441=1134.179,-26.643,-48.169,179.320,6.253,149.332
C02442=1134.174,-26.394,-48.182,179.322,6.254,149.332
C02443=1134.169,-26.144,-48.194,179.324,6.254,149.331
C02444=1134.163,-25.894,-48.205,179.327,6.255,149.330
C02445=1134.158,-25.645,-48.217,179.329,6.256,149.330
C02446=1134.153,-25.395,-48.229,179.331,6.256,149.329
C02447=1134.147,-25.126,-48.242,179.334,6.258,149.329
C02448=1134.142,-24.855,-48.255,179.337,6.258,149.328
C02449=1134.136,-24.585,-48.268,179.339,6.259,149.328
C02450=1134.130,-24.315,-48.281,179.342,6.259,149.327
C02451=1134.125,-24.065,-48.293,179.344,6.260,149.326
C02452=1134.120,-23.816,-48.305,179.346,6.261,149.326
C02453=1134.115,-23.566,-48.317,179.348,6.262,149.325
C02454=1134.110,-23.316,-48.329,179.352,6.263,149.325
C02455=1134.104,-23.067,-48.341,179.354,6.264,149.324
C02456=1134.099,-22.817,-48.353,179.356,6.264,149.324
C02457=1134.094,-22.567,-48.365,179.359,6.265,149.323
C02458=1134.088,-22.318,-48.378,179.361,6.266,149.323
C02459=1134.084,-22.068,-48.389,179.363,6.266,149.322
C02460=1134.079,-21.819,-48.402,179.366,6.267,149.321
C02461=1134.073,-21.569,-48.413,179.368,6.268,149.321
C02462=1134.068,-21.320,-48.426,179.370,6.268,149.321
C02463=1134.063,-21.070,-48.438,179.373,6.269,149.320
C02464=1134.057,-20.820,-48.450,179.375,6.270,149.319
C02465=1134.052,-20.570,-48.462,179.378,6.271,149.319
C02466=1134.047,-20.320,-48.474,179.380,6.271,149.318
C02467=1134.042,-20.071,-48.487,179.382,6.272,149.318
C02468=1134.036,-19.821,-48.499,179.385,6.273,149.317
C02469=1134.031,-19.572,-48.511,179.387,6.273,149.317
C02470=1134.026,-19.322,-48.523,179.389,6.274,149.316
C02471=1134.021,-19.073,-48.535,179.392,6.275,149.316
C02472=1134.016,-18.822,-48.548,179.394,6.275,149.315
C02473=1134.011,-18.573,-48.560,179.397,6.276,149.314
C02474=1134.006,-18.323,-48.572,179.399,6.278,149.314
C02475=1134.001,-18.074,-48.585,179.402,6.278,149.313
C02476=1133.995,-17.824,-48.597,179.404,6.279,149.313
C02477=1133.990,-17.574,-48.609,179.406,6.280,149.312
C02478=1133.985,-17.324,-48.621,179.409,6.281,149.312
C02479=1133.980,-17.075,-48.634,179.411,6.281,149.311
C02480=1133.974,-16.826,-48.646,179.413,6.282,149.311
C02481=1133.969,-16.576,-48.658,179.416,6.283,149.310
C02482=1133.964,-16.327,-48.671,179.419,6.284,149.310
C02483=1133.958,-16.077,-48.683,179.421,6.285,149.309
C02484=1133.954,-15.827,-48.696,179.423,6.285,149.309
C02485=1133.949,-15.577,-48.708,179.426,6.286,149.308
C02486=1133.943,-15.327,-48.720,179.428,6.287,149.307
C02487=1133.938,-15.078,-48.733,179.430,6.287,149.307
C02488=1133.933,-14.829,-48.745,179.433,6.288,149.306
C02489=1133.928,-14.579,-48.757,179.435,6.289,149.306
C02490=1133.923,-14.329,-48.770,179.438,6.290,149.305
C02491=1133.917,-14.080,-48.783,179.440,6.291,149.305
C02492=1133.912,-13.829,-48.795,179.443,6.291,149.304
C02493=1133.907,-13.580,-48.808,179.445,6.292,149.304
C02494=1133.902,-13.331,-48.820,179.447,6.293,149.303
C02495=1133.896,-13.081,-48.832,179.450,6.293,149.303
C02496=1133.891,-12.831,-48.845,179.452,6.295,149.302
C02497=1133.886,-12.582,-48.857,179.455,6.295,149.301
C02498=1133.880,-12.332,-48.869,179.457,6.296,149.301
C02499=1133.876,-12.082,-48.882,179.459,6.297,149.300
C02500=1133.871,-11.833,-48.895,179.462,6.297,149.300
C02501=1133.866,-11.583,-48.908,179.464,6.298,149.299
C02502=1133.860,-11.333,-48.920,179.467,6.299,149.299
C02503=1133.854,-11.084,-48.933,179.470,6.300,149.298
C02504=1133.850,-10.834,-48.946,179.472,6.301,149.298
C02505=1133.845,-10.585,-48.958,179.474,6.302,149.297
C02506=1133.840,-10.335,-48.971,179.477,6.302,149.296
C02507=1133.834,-10.085,-48.983,179.479,6.303,149.296
C02508=1133.829,-9.836,-48.995,179.481,6.304,149.296
C02509=1133.825,-9.586,-49.008,179.484,6.305,149.295
C02510=1133.819,-9.336,-49.021,179.487,6.306,149.294
C02511=1133.814,-9.087,-49.034,179.489,6.307,149.294
C02512=1133.808,-8.838,-49.047,179.491,6.307,149.293
C02513=1133.804,-8.587,-49.059,179.494,6.308,149.293
C02514=1133.799,-8.338,-49.071,179.496,6.309,149.292
C02515=1133.793,-8.088,-49.085,179.499,6.310,149.292
C02516=1133.788,-7.839,-49.097,179.501,6.311,149.291
C02517=1133.782,-7.589,-49.110,179.503,6.311,149.291
C02518=1133.778,-7.339,-49.123,179.506,6.312,149.290
C02519=1133.773,-7.090,-49.135,179.508,6.313,149.289
C02520=1133.767,-6.840,-49.149,179.511,6.314,149.289
C02521=1133.762,-6.591,-49.161,179.514,6.315,149.288
C02522=1133.757,-6.341,-49.174,179.516,6.315,149.288
C02523=1133.752,-6.091,-49.186,179.518,6.316,149.287
C02524=1133.746,-5.842,-49.199,179.521,6.317,149.287
C02525=1133.741,-5.592,-49.212,179.523,6.318,149.286
C02526=1133.736,-5.342,-49.225,179.526,6.319,149.286
C02527=1133.731,-5.093,-49.237,179.528,6.319,149.285
C02528=1133.725,-4.843,-49.251,179.531,6.320,149.285
C02529=1133.721,-4.593,-49.264,179.533,6.321,149.284
C02530=1133.716,-4.344,-49.276,179.536,6.322,149.283
C02531=1133.710,-4.094,-49.289,179.538,6.323,149.283
C02532=1133.705,-3.844,-49.302,179.540,6.324,149.282
C02533=1133.700,-3.595,-49.315,179.543,6.324,149.282
C02534=1133.694,-3.345,-49.328,179.545,6.325,149.281
C02535=1133.690,-3.095,-49.341,179.548,6.327,149.281
C02536=1133.685,-2.846,-49.354,179.551,6.327,149.280
C02537=1133.679,-2.597,-49.368,179.553,6.328,149.280
C02538=1133.674,-2.348,-49.380,179.555,6.329,149.279
C02539=1133.669,-2.098,-49.393,179.558,6.330,149.279
C02540=1133.664,-1.848,-49.406,179.560,6.331,149.278
C02541=1133.658,-1.599,-49.419,179.563,6.331,149.278
C02542=1133.654,-1.349,-49.432,179.565,6.332,149.277
C02543=1133.648,-1.099,-49.445,179.567,6.333,149.276
C02544=1133.643,-0.850,-49.458,179.570,6.334,149.276
C02545=1133.638,-0.600,-49.471,179.573,6.335,149.275
C02546=1133.633,-0.350,-49.484,179.575,6.335,149.275
C02547=1133.628,-0.101,-49.498,179.577,6.336,149.274
C02548=1133.623,0.149,-49.511,179.580,6.337,149.274
C02549=1133.617,0.398,-49.523,179.583,6.338,149.273
C02550=1133.612,0.649,-49.537,179.585,6.339,149.273
C02551=1133.607,0.918,-49.550,179.588,6.340,149.272
C02552=1133.601,1.187,-49.565,179.590,6.341,149.272
C02553=1133.596,1.457,-49.579,179.593,6.341,149.271
C02554=1133.590,1.726,-49.593,179.596,6.343,149.270
C02555=1133.585,1.976,-49.607,179.598,6.343,149.270
C02556=1133.580,2.225,-49.620,179.600,6.344,149.269
C02557=1133.575,2.475,-49.633,179.603,6.346,149.269
C02558=1133.569,2.725,-49.646,179.606,6.346,149.268
C02559=1133.564,2.973,-49.659,179.608,6.347,149.268
C02560=1133.559,3.224,-49.673,179.610,6.348,149.267
C02561=1133.554,3.473,-49.685,179.614,6.349,149.267
C02562=1133.549,3.723,-49.699,179.616,6.350,149.266
C02563=1133.544,3.972,-49.712,179.618,6.351,149.266
C02564=1133.539,4.222,-49.726,179.621,6.351,149.265
C02565=1133.534,4.472,-49.738,179.623,6.353,149.264
C02566=1133.529,4.721,-49.753,179.626,6.354,149.264
C02567=1133.524,4.971,-49.765,179.628,6.354,149.263
C02568=1133.518,5.220,-49.779,179.630,6.355,149.263
C02569=1133.513,5.470,-49.792,179.633,6.356,149.262
C02570=1133.508,5.719,-49.805,179.636,6.357,149.262
C02571=1133.503,5.969,-49.818,179.638,6.358,149.261
C02572=1133.498,6.218,-49.832,179.641,6.359,149.261
C02573=1133.492,6.469,-49.846,179.643,6.360,149.260
C02574=1133.487,6.717,-49.859,179.646,6.360,149.260
C02575=1133.482,6.968,-49.873,179.648,6.361,149.259
C02576=1133.477,7.217,-49.885,179.651,6.362,149.258
C02577=1133.472,7.467,-49.900,179.653,6.363,149.258
C02578=1133.467,7.716,-49.912,179.655,6.364,149.258
C02579=1133.462,7.966,-49.926,179.659,6.365,149.257
C02580=1133.456,8.216,-49.940,179.661,6.366,149.256
C02581=1133.452,8.466,-49.953,179.663,6.367,149.256
C02582=1133.446,8.715,-49.967,179.666,6.367,149.255
C02583=1133.441,8.965,-49.980,179.668,6.369,149.255
C02584=1133.436,9.214,-49.993,179.671,6.370,149.254
C02585=1133.431,9.464,-50.007,179.673,6.370,149.254
C02586=1133.426,9.713,-50.020,179.676,6.372,149.253
C02587=1133.421,9.963,-50.034,179.678,6.373,149.253
C02588=1133.415,10.212,-50.048,179.681,6.373,149.252
C02589=1133.411,10.462,-50.061,179.684,6.375,149.252
C02590=1133.405,10.711,-50.075,179.686,6.375,149.251
C02591=1133.400,10.961,-50.088,179.688,6.376,149.250
C02592=1133.396,11.211,-50.102,179.691,6.377,149.250
C02593=1133.390,11.460,-50.116,179.693,6.378,149.249
C02594=1133.385,11.710,-50.129,179.696,6.379,149.249
C02595=1133.380,11.959,-50.143,179.698,6.379,149.248
C02596=1133.375,12.209,-50.156,179.701,6.381,149.248
C02597=1133.369,12.458,-50.170,179.704,6.382,149.247
C02598=1133.364,12.708,-50.184,179.706,6.382,149.247
C02599=1133.360,12.958,-50.197,179.709,6.384,149.246
C02600=1133.354,13.207,-50.211,179.711,6.384,149.246
C02601=1133.349,13.457,-50.225,179.713,6.385,149.245
C02602=1133.343,13.706,-50.239,179.716,6.387,149.245
C02603=1133.339,13.956,-50.252,179.719,6.387,149.244
C02604=1133.333,14.205,-50.266,179.721,6.388,149.244
C02605=1133.328,14.455,-50.280,179.724,6.390,149.243
C02606=1133.323,14.705,-50.294,179.726,6.390,149.242
C02607=1133.318,14.954,-50.307,179.729,6.391,149.242
C02608=1133.313,15.204,-50.321,179.731,6.392,149.241
C02609=1133.308,15.453,-50.335,179.734,6.393,149.241
C02610=1133.302,15.703,-50.349,179.736,6.394,149.240
C02611=1133.298,15.952,-50.362,179.739,6.395,149.240
C02612=1133.293,16.201,-50.376,179.742,6.396,149.239
C02613=1133.288,16.451,-50.390,179.744,6.397,149.239
C02614=1133.282,16.701,-50.404,179.747,6.398,149.238
C02615=1133.277,16.950,-50.418,179.749,6.399,149.238
C02616=1133.272,17.200,-50.432,179.752,6.400,149.237
C02617=1133.268,17.450,-50.446,179.754,6.401,149.237
C02618=1133.262,17.699,-50.459,179.757,6.401,149.236
C02619=1133.257,17.949,-50.473,179.760,6.403,149.235
C02620=1133.252,18.199,-50.488,179.762,6.404,149.235
C02621=1133.246,18.448,-50.502,179.764,6.404,149.234
C02622=1133.241,18.697,-50.516,179.767,6.406,149.234
C02623=1133.236,18.948,-50.529,179.769,6.407,149.233
C02624=1133.231,19.196,-50.543,179.772,6.408,149.233
C02625=1133.226,19.446,-50.557,179.775,6.409,149.232
C02626=1133.221,19.696,-50.571,179.777,6.410,149.232
C02627=1133.216,19.945,-50.586,179.780,6.411,149.231
C02628=1133.211,20.194,-50.599,179.782,6.412,149.231
C02629=1133.206,20.444,-50.614,179.785,6.412,149.230
C02630=1133.201,20.695,-50.627,179.787,6.414,149.230
C02631=1133.195,20.944,-50.641,179.790,6.414,149.229
C02632=1133.190,21.193,-50.655,179.792,6.415,149.229
C02633=1133.185,21.443,-50.670,179.795,6.417,149.228
C02634=1133.180,21.693,-50.684,179.798,6.417,149.228
C02635=1133.175,21.942,-50.698,179.800,6.419,149.227
C02636=1133.170,22.191,-50.712,179.802,6.420,149.227
C02637=1133.166,22.441,-50.726,179.805,6.420,149.226
C02638=1133.161,22.690,-50.740,179.808,6.422,149.225
C02639=1133.155,22.939,-50.754,179.810,6.423,149.225
C02640=1133.150,23.189,-50.768,179.813,6.424,149.224
C02641=1133.145,23.439,-50.783,179.816,6.425,149.224
C02642=1133.140,23.689,-50.797,179.818,6.425,149.223
C02643=1133.135,23.938,-50.811,179.821,6.427,149.223
C02644=1133.130,24.187,-50.825,179.823,6.428,149.222
C02645=1133.125,24.437,-50.839,179.826,6.429,149.222
C02646=1133.120,24.687,-50.854,179.829,6.430,149.221
C02647=1133.115,24.936,-50.868,179.831,6.430,149.221
C02648=1133.109,25.185,-50.882,179.833,6.432,149.220
C02649=1133.104,25.436,-50.897,179.836,6.432,149.220
C02650=1133.099,25.685,-50.911,179.839,6.434,149.219
C02651=1133.094,25.935,-50.925,179.841,6.435,149.219
C02652=1133.089,26.185,-50.940,179.844,6.435,149.218
C02653=1133.083,26.433,-50.954,179.846,6.437,149.217
C02654=1133.078,26.683,-50.968,179.849,6.438,149.217
C02655=1133.073,26.952,-50.983,179.852,6.439,149.216
C02656=1133.068,27.221,-50.999,179.855,6.441,149.216
C02657=1133.062,27.490,-51.014,179.857,6.441,149.215
C02658=1133.057,27.759,-51.030,179.860,6.443,149.215
C02659=1133.051,28.008,-51.044,179.862,6.443,149.214
C02660=1133.046,28.258,-51.059,179.865,6.445,149.214
C02661=1133.041,28.507,-51.074,179.868,6.446,149.213
C02662=1133.036,28.757,-51.088,179.870,6.446,149.213
C02663=1133.032,29.007,-51.102,179.873,6.448,149.212
C02664=1133.027,29.256,-51.116,179.875,6.448,149.212
C02665=1133.021,29.506,-51.131,179.878,6.450,149.211
C02666=1133.016,29.755,-51.146,179.881,6.450,149.210
C02667=1133.011,30.005,-51.160,179.883,6.452,149.210
C02668=1133.006,30.254,-51.174,179.886,6.453,149.210
C02669=1133.001,30.504,-51.189,179.889,6.454,149.209
C02670=1132.996,30.753,-51.204,179.891,6.455,149.208
C02671=1132.990,31.003,-51.219,179.894,6.457,149.208
C02672=1132.985,31.253,-51.233,179.896,6.457,149.207
C02673=1132.981,31.502,-51.247,179.899,6.458,149.207
C02674=1132.976,31.752,-51.262,179.901,6.459,149.206
C02675=1132.971,32.001,-51.276,179.904,6.460,149.206
C02676=1132.965,32.251,-51.291,179.907,6.461,149.205
C02677=1132.960,32.500,-51.306,179.909,6.462,149.205
C02678=1132.955,32.749,-51.320,179.912,6.464,149.204
C02679=1132.950,32.999,-51.335,179.914,6.464,149.204
C02680=1132.945,33.249,-51.350,179.917,6.466,149.203
C02681=1132.940,33.498,-51.364,179.919,6.467,149.203
C02682=1132.935,33.748,-51.379,179.923,6.468,149.202
C02683=1132.930,33.997,-51.394,179.925,6.469,149.202
C02684=1132.924,34.247,-51.409,179.927,6.470,149.201
C02685=1132.920,34.496,-51.424,179.930,6.471,149.200
C02686=1132.915,34.746,-51.438,179.932,6.472,149.200
C02687=1132.910,34.996,-51.452,179.935,6.473,149.200
C02688=1132.904,35.245,-51.468,179.937,6.474,149.199
C02689=1132.900,35.495,-51.482,179.940,6.475,149.198
C02690=1132.895,35.744,-51.497,179.943,6.476,149.198
C02691=1132.889,35.994,-51.512,179.945,6.478,149.198
C02692=1132.885,36.243,-51.527,179.948,6.478,149.197
C02693=1132.880,36.493,-51.541,179.951,6.480,149.196
C02694=1132.874,36.742,-51.557,179.953,6.481,149.196
C02695=1132.869,36.992,-51.571,179.956,6.482,149.195
C02696=1132.865,37.241,-51.586,179.958,6.483,149.195
C02697=1132.859,37.491,-51.601,179.961,6.484,149.194
C02698=1132.854,37.740,-51.616,179.964,6.485,149.194
C02699=1132.849,37.990,-51.631,179.967,6.487,149.193
C02700=1132.844,38.239,-51.646,179.969,6.487,149.193
C02701=1132.839,38.489,-51.660,179.971,6.489,149.192
C02702=1132.834,38.738,-51.676,179.974,6.489,149.192
C02703=1132.829,38.987,-51.691,179.977,6.491,149.191
C02704=1132.823,39.237,-51.705,179.979,6.492,149.191
C02705=1132.819,39.486,-51.720,179.982,6.493,149.190
C02706=1132.814,39.736,-51.735,179.984,6.494,149.190
C02707=1132.808,39.985,-51.750,179.987,6.496,149.189
C02708=1132.804,40.235,-51.765,179.990,6.496,149.189
C02709=1132.798,40.485,-51.780,179.993,6.498,149.188
C02710=1132.793,40.734,-51.795,179.995,6.499,149.188
C02711=1132.788,40.983,-51.811,179.998,6.500,149.187
C02712=1132.783,41.233,-51.825,-179.999,6.501,149.187
C02713=1132.778,41.482,-51.841,-179.997,6.502,149.186
C02714=1132.773,41.731,-51.856,-179.994,6.504,149.186
C02715=1132.767,41.981,-51.870,-179.992,6.504,149.185
C02716=1132.763,42.231,-51.886,-179.989,6.506,149.185
C02717=1132.758,42.480,-51.901,-179.987,6.507,149.184
C02718=1132.753,42.730,-51.916,-179.984,6.508,149.184
C02719=1132.747,42.980,-51.931,-179.981,6.509,149.183
C02720=1132.743,43.229,-51.946,-179.979,6.510,149.183
C02721=1132.737,43.478,-51.962,-179.976,6.511,149.182
C02722=1132.732,43.728,-51.976,-179.973,6.512,149.181
C02723=1132.727,43.977,-51.992,-179.970,6.514,149.181
C02724=1132.722,44.226,-52.007,-179.968,6.515,149.180
C02725=1132.718,44.476,-52.023,-179.965,6.516,149.180
C02726=1132.713,44.726,-52.037,-179.963,6.517,149.179
C02727=1132.707,44.975,-52.052,-179.960,6.519,149.179
C02728=1132.703,45.225,-52.067,-179.958,6.519,149.178
C02729=1132.697,45.474,-52.083,-179.955,6.521,149.178
C02730=1132.692,45.723,-52.099,-179.952,6.522,149.177
C02731=1132.687,45.972,-52.114,-179.950,6.523,149.177
C02732=1132.682,46.223,-52.129,-179.946,6.524,149.176
C02733=1132.677,46.472,-52.144,-179.944,6.525,149.176
C02734=1132.672,46.722,-52.159,-179.942,6.527,149.175
C02735=1132.667,46.971,-52.175,-179.939,6.528,149.175
C02736=1132.662,47.220,-52.190,-179.936,6.529,149.174
C02737=1132.657,47.470,-52.206,-179.934,6.530,149.174
C02738=1132.653,47.719,-52.221,-179.931,6.531,149.173
C02739=1132.647,47.969,-52.237,-179.929,6.532,149.173
C02740=1132.642,48.218,-52.252,-179.926,6.533,149.172
C02741=1132.637,48.467,-52.267,-179.923,6.535,149.172
C02742=1132.632,48.717,-52.283,-179.921,6.536,149.171
C02743=1132.627,48.967,-52.299,-179.918,6.537,149.171
C02744=1132.622,49.216,-52.314,-179.915,6.538,149.170
C02745=1132.617,49.465,-52.329,-179.913,6.540,149.170
C02746=1132.612,49.715,-52.345,-179.910,6.541,149.169
C02747=1132.607,49.964,-52.360,-179.907,6.542,149.169
C02748=1132.602,50.214,-52.376,-179.905,6.543,149.168
C02749=1132.597,50.463,-52.391,-179.902,6.544,149.168
C02750=1132.592,50.712,-52.406,-179.899,6.545,149.167
C02751=1132.587,50.962,-52.422,-179.896,6.547,149.167
C02752=1132.582,51.212,-52.438,-179.894,6.548,149.166
C02753=1132.577,51.461,-52.454,-179.891,6.550,149.166
C02754=1132.572,51.711,-52.469,-179.889,6.550,149.165
C02755=1132.567,51.960,-52.484,-179.886,6.552,149.165
C02756=1132.562,52.210,-52.500,-179.883,6.553,149.164
C02757=1132.556,52.459,-52.516,-179.881,6.554,149.164
C02758=1132.552,52.709,-52.531,-179.878,6.555,149.163
C02759=1132.547,52.978,-52.548,-179.875,6.557,149.163
C02760=1132.541,53.246,-52.565,-179.872,6.557,149.162
C02761=1132.536,53.515,-52.582,-179.870,6.559,149.162
C02762=1132.530,53.783,-52.599,-179.866,6.560,149.161
C02763=1132.525,54.033,-52.615,-179.864,6.562,149.160
C02764=1132.520,54.283,-52.631,-179.862,6.563,149.160
C02765=1132.515,54.532,-52.646,-179.859,6.564,149.160
C02766=1132.510,54.781,-52.661,-179.856,6.566,149.159
C02767=1132.505,55.030,-52.678,-179.853,6.567,149.158
C02768=1132.500,55.280,-52.693,-179.851,6.568,149.158
C02769=1132.495,55.529,-52.709,-179.848,6.569,149.158
C02770=1132.490,55.779,-52.725,-179.845,6.570,149.157
C02771=1132.485,56.028,-52.740,-179.842,6.572,149.156
C02772=1132.480,56.277,-52.756,-179.840,6.573,149.156
C02773=1132.475,56.527,-52.772,-179.838,6.574,149.156
C02774=1132.470,56.777,-52.788,-179.834,6.576,149.155
C02775=1132.465,57.027,-52.804,-179.832,6.576,149.154
C02776=1132.460,57.276,-52.820,-179.829,6.578,149.154
C02777=1132.455,57.525,-52.836,-179.827,6.580,149.154
C02778=1132.450,57.775,-52.852,-179.824,6.580,149.153
C02779=1132.445,58.024,-52.868,-179.821,6.582,149.152
C02780=1132.439,58.273,-52.884,-179.819,6.583,149.152
C02781=1132.435,58.523,-52.899,-179.816,6.584,149.152
C02782=1132.430,58.772,-52.915,-179.813,6.586,149.151
C02783=1132.425,59.022,-52.931,-179.811,6.586,149.150
C02784=1132.420,59.271,-52.947,-179.808,6.588,149.150
C02785=1132.415,59.520,-52.963,-179.805,6.590,149.150
C02786=1132.410,59.770,-52.979,-179.803,6.590,149.149
C02787=1132.405,60.019,-52.995,-179.800,6.592,149.149
C02788=1132.400,60.269,-53.011,-179.797,6.593,149.148
C02789=1132.395,60.518,-53.028,-179.795,6.594,149.148
C02790=1132.390,60.767,-53.043,-179.792,6.596,149.147
C02791=1132.385,61.017,-53.059,-179.789,6.597,149.147
C02792=1132.380,61.266,-53.075,-179.787,6.598,149.146
C02793=1132.375,61.516,-53.091,-179.784,6.600,149.146
C02794=1132.370,61.765,-53.108,-179.781,6.601,149.145
C02795=1132.365,62.015,-53.124,-179.778,6.603,149.145
C02796=1132.360,62.264,-53.140,-179.776,6.603,149.144
C02797=1132.355,62.514,-53.156,-179.773,6.605,149.144
C02798=1132.350,62.763,-53.172,-179.770,6.606,149.143
C02799=1132.346,63.013,-53.188,-179.768,6.607,149.143
C02800=1132.341,63.262,-53.204,-179.765,6.609,149.142
C02801=1132.335,63.512,-53.221,-179.762,6.610,149.142
C02802=1132.330,63.761,-53.237,-179.760,6.611,149.141
C02803=1132.325,64.010,-53.254,-179.757,6.613,149.141
C02804=1132.320,64.260,-53.270,-179.754,6.614,149.140
C02805=1132.316,64.509,-53.286,-179.752,6.615,149.140
C02806=1132.310,64.759,-53.302,-179.749,6.616,149.139
C02807=1132.306,65.008,-53.318,-179.746,6.618,149.139
C02808=1132.301,65.257,-53.335,-179.743,6.620,149.138
C02809=1132.296,65.507,-53.351,-179.741,6.620,149.138
C02810=1132.291,65.756,-53.367,-179.738,6.622,149.137
C02811=1132.285,66.006,-53.384,-179.735,6.623,149.137
C02812=1132.280,66.255,-53.400,-179.733,6.624,149.136
C02813=1132.276,66.505,-53.417,-179.730,6.626,149.136
C02814=1132.270,66.754,-53.432,-179.728,6.627,149.135
C02815=1132.266,67.004,-53.449,-179.724,6.629,149.135
C02816=1132.261,67.252,-53.465,-179.722,6.630,149.134
C02817=1132.256,67.502,-53.482,-179.719,6.631,149.134
C02818=1132.251,67.752,-53.498,-179.717,6.633,149.133
C02819=1132.246,68.001,-53.515,-179.714,6.633,149.133
C02820=1132.241,68.250,-53.531,-179.711,6.635,149.132
C02821=1132.236,68.500,-53.547,-179.709,6.637,149.132
C02822=1132.231,68.750,-53.564,-179.706,6.638,149.131
C02823=1132.225,68.998,-53.580,-179.704,6.639,149.131
C02824=1132.221,69.248,-53.597,-179.700,6.640,149.130
C02825=1132.217,69.497,-53.614,-179.698,6.642,149.130
C02826=1132.210,69.747,-53.630,-179.695,6.644,149.129
C02827=1132.206,69.997,-53.647,-179.693,6.644,149.129
C02828=1132.201,70.245,-53.663,-179.690,6.646,149.128
C02829=1132.196,70.495,-53.680,-179.687,6.647,149.128
C02830=1132.191,70.745,-53.697,-179.684,6.649,149.127
C02831=1132.186,70.993,-53.713,-179.682,6.650,149.127
C02832=1132.181,71.244,-53.729,-179.679,6.652,149.127
C02833=1132.177,71.493,-53.746,-179.676,6.653,149.126
C02834=1132.171,71.742,-53.763,-179.673,6.654,149.126
C02835=1132.166,71.992,-53.779,-179.671,6.655,149.125
C02836=1132.161,72.240,-53.796,-179.668,6.657,149.125
C02837=1132.156,72.490,-53.813,-179.665,6.658,149.124
C02838=1132.152,72.740,-53.830,-179.662,6.660,149.124
C02839=1132.147,72.988,-53.846,-179.660,6.661,149.123
C02840=1132.141,73.238,-53.863,-179.657,6.662,149.123
C02841=1132.137,73.488,-53.880,-179.655,6.664,149.122
C02842=1132.132,73.737,-53.896,-179.651,6.665,149.122
C02843=1132.127,73.986,-53.913,-179.649,6.666,149.121
C02844=1132.122,74.236,-53.930,-179.646,6.668,149.121
C02845=1132.116,74.485,-53.947,-179.644,6.669,149.120
C02846=1132.112,74.734,-53.964,-179.641,6.671,149.120
C02847=1132.107,74.984,-53.980,-179.638,6.672,149.119
C02848=1132.102,75.234,-53.998,-179.636,6.673,149.119
C02849=1132.097,75.482,-54.014,-179.633,6.675,149.118
C02850=1132.092,75.732,-54.031,-179.630,6.676,149.118
C02851=1132.087,75.982,-54.048,-179.627,6.678,149.118
C02852=1132.082,76.230,-54.064,-179.625,6.679,149.117
C02853=1132.077,76.480,-54.081,-179.622,6.680,149.116
C02854=1132.073,76.730,-54.098,-179.619,6.682,149.116
C02855=1132.067,76.980,-54.115,-179.616,6.684,149.116
C02856=1132.062,77.228,-54.132,-179.614,6.685,149.115
C02857=1132.057,77.478,-54.149,-179.611,6.686,149.114
C02858=1132.053,77.728,-54.166,-179.608,6.687,149.114
C02859=1132.048,77.977,-54.184,-179.606,6.689,149.114
C02860=1132.043,78.226,-54.200,-179.603,6.691,149.113
C02861=1132.037,78.475,-54.217,-179.600,6.692,149.113
C02862=1132.033,78.725,-54.234,-179.598,6.693,149.112
C02863=1132.027,78.993,-54.252,-179.595,6.694,149.112
C02864=1132.022,79.262,-54.270,-179.592,6.696,149.111
C02865=1132.017,79.530,-54.289,-179.588,6.698,149.111
C02866=1132.011,79.799,-54.307,-179.585,6.700,149.110
C02867=1132.007,80.048,-54.325,-179.583,6.701,149.110
C02868=1132.001,80.297,-54.342,-179.580,6.702,149.109
C02869=1131.997,80.547,-54.359,-179.578,6.704,149.109
C02870=1131.991,80.796,-54.375,-179.574,6.705,149.108
C02871=1131.987,81.045,-54.393,-179.572,6.707,149.108
C02872=1131.982,81.295,-54.410,-179.570,6.708,149.107
C02873=1131.977,81.544,-54.427,-179.567,6.709,149.107
C02874=1131.972,81.794,-54.444,-179.564,6.711,149.107
C02875=1131.967,82.043,-54.462,-179.561,6.713,149.106
C02876=1131.962,82.292,-54.478,-179.558,6.714,149.105
C02877=1131.957,82.542,-54.496,-179.555,6.716,149.105
C02878=1131.952,82.791,-54.514,-179.553,6.716,149.105
C02879=1131.948,83.040,-54.530,-179.550,6.718,149.104
C02880=1131.942,83.290,-54.547,-179.548,6.720,149.104
C02881=1131.937,83.539,-54.565,-179.545,6.721,149.103
C02882=1131.933,83.789,-54.582,-179.542,6.723,149.103
C02883=1131.927,84.037,-54.600,-179.539,6.724,149.102
C02884=1131.922,84.287,-54.617,-179.536,6.726,149.102
C02885=1131.918,84.536,-54.634,-179.534,6.727,149.101
C02886=1131.913,84.786,-54.652,-179.531,6.729,149.101
C02887=1131.908,85.035,-54.669,-179.529,6.730,149.101
C02888=1131.903,85.284,-54.686,-179.525,6.731,149.100
C02889=1131.898,85.534,-54.704,-179.523,6.733,149.099
C02890=1131.893,85.783,-54.722,-179.520,6.735,149.099
C02891=1131.889,86.033,-54.738,-179.517,6.736,149.099
C02892=1131.883,86.281,-54.756,-179.515,6.737,149.098
C02893=1131.878,86.531,-54.773,-179.512,6.739,149.098
C02894=1131.873,86.780,-54.791,-179.509,6.740,149.097
C02895=1131.869,87.030,-54.808,-179.506,6.742,149.097
C02896=1131.864,87.279,-54.826,-179.504,6.744,149.096
C02897=1131.859,87.529,-54.843,-179.501,6.745,149.096
C02898=1131.854,87.778,-54.861,-179.498,6.747,149.095
C02899=1131.849,88.027,-54.878,-179.495,6.748,149.095
C02900=1131.844,88.276,-54.896,-179.493,6.749,149.095
C02901=1131.839,88.526,-54.914,-179.490,6.751,149.094
C02902=1131.834,88.775,-54.931,-179.487,6.752,149.093
C02903=1131.829,89.025,-54.949,-179.484,6.754,149.093
C02904=1131.825,89.274,-54.966,-179.482,6.756,149.093
C02905=1131.820,89.523,-54.983,-179.479,6.757,149.092
C02906=1131.815,89.772,-55.001,-179.476,6.759,149.092
C02907=1131.810,90.022,-55.019,-179.473,6.760,149.091
C02908=1131.805,90.271,-55.037,-179.470,6.762,149.091
C02909=1131.800,90.521,-55.055,-179.468,6.763,149.090
C02910=1131.795,90.770,-55.071,-179.465,6.764,149.090
C02911=1131.790,91.019,-55.089,-179.463,6.766,149.089
C02912=1131.786,91.268,-55.107,-179.460,6.768,149.089
C02913=1131.781,91.518,-55.125,-179.457,6.769,149.089
C02914=1131.775,91.767,-55.143,-179.454,6.771,149.088
C02915=1131.770,92.017,-55.161,-179.451,6.772,149.088
C02916=1131.766,92.266,-55.179,-179.448,6.774,149.087
C02917=1131.761,92.515,-55.196,-179.446,6.776,149.087
C02918=1131.755,92.765,-55.214,-179.443,6.777,149.086
C02919=1131.751,93.014,-55.231,-179.440,6.779,149.086
C02920=1131.746,93.263,-55.249,-179.438,6.780,149.085
C02921=1131.741,93.512,-55.267,-179.435,6.781,149.085
C02922=1131.737,93.761,-55.285,-179.433,6.783,149.085
C02923=1131.731,94.011,-55.302,-179.429,6.784,149.084
C02924=1131.726,94.260,-55.320,-179.427,6.786,149.084
C02925=1131.721,94.509,-55.338,-179.424,6.788,149.083
C02926=1131.717,94.758,-55.356,-179.421,6.789,149.083
C02927=1131.712,95.008,-55.374,-179.418,6.791,149.082
C02928=1131.707,95.257,-55.393,-179.416,6.793,149.082
C02929=1131.702,95.507,-55.411,-179.413,6.794,149.081
C02930=1131.697,95.756,-55.428,-179.410,6.796,149.081
C02931=1131.692,96.006,-55.446,-179.407,6.797,149.080
C02932=1131.687,96.255,-55.464,-179.404,6.799,149.080
C02933=1131.682,96.504,-55.482,-179.401,6.801,149.080
C02934=1131.678,96.753,-55.500,-179.399,6.802,149.079
C02935=1131.673,97.002,-55.518,-179.396,6.804,149.079
C02936=1131.668,97.252,-55.536,-179.394,6.805,149.078
C02937=1131.663,97.501,-55.554,-179.391,6.807,149.078
C02938=1131.658,97.751,-55.573,-179.388,6.808,149.077
C02939=1131.653,97.995,-55.590,-179.386,6.810,149.077
C02940=1131.648,98.240,-55.607,-179.383,6.812,149.077
C02941=1131.643,98.485,-55.626,-179.380,6.813,149.076
C02942=1131.620,99.706,-55.713,-179.975,7.965,149.508
C02943=1131.615,99.954,-55.732,-179.974,7.969,149.509
C02944=1131.610,100.205,-55.751,-179.971,7.973,149.509
C02945=1131.605,100.454,-55.769,-179.969,7.977,149.509
C02946=1131.600,100.703,-55.787,-179.967,7.981,149.509
C02947=1131.595,100.951,-55.805,-179.965,7.985,149.510
C02948=1131.590,101.202,-55.824,-179.963,7.989,149.510
C02949=1131.586,101.451,-55.842,-179.961,7.993,149.511
C02950=1131.581,101.699,-55.861,-179.959,7.997,149.511
C02951=1131.576,101.950,-55.880,-179.957,8.002,149.511
C02952=1131.571,102.199,-55.898,-179.954,8.005,149.511
C02953=1131.566,102.447,-55.917,-179.952,8.009,149.512
C02954=1131.561,102.698,-55.936,-179.950,8.013,149.512
C02955=1131.555,103.019,-55.959,-179.947,8.018,149.512
C02956=1131.549,103.342,-55.983,-179.944,8.024,149.513
C02957=1131.542,103.664,-56.007,-179.941,8.029,149.513
C02958=1131.536,103.987,-56.032,-179.938,8.034,149.513
C02959=1131.532,104.236,-56.050,-179.936,8.038,149.514
C02960=1131.527,104.485,-56.069,-179.934,8.042,149.514
C02961=1131.522,104.735,-56.087,-179.931,8.046,149.514
C02962=1131.517,104.983,-56.106,-179.929,8.050,149.514
C02963=1131.512,105.233,-56.126,-179.927,8.054,149.515
C02964=1131.507,105.482,-56.144,-179.924,8.058,149.515
C02965=1131.502,105.731,-56.163,-179.922,8.063,149.515
C02966=1131.498,105.981,-56.181,-179.920,8.066,149.515
C02967=1131.493,106.229,-56.200,-179.917,8.070,149.516
C02968=1131.488,106.480,-56.219,-179.915,8.074,149.516
C02969=1131.483,106.728,-56.238,-179.912,8.078,149.516
C02970=1131.479,106.978,-56.257,-179.910,8.082,149.516
C02971=1131.474,107.227,-56.275,-179.908,8.086,149.517
C02972=1131.468,107.476,-56.295,-179.905,8.090,149.517
C02973=1131.464,107.725,-56.314,-179.902,8.094,149.517
C02974=1131.459,107.975,-56.332,-179.900,8.098,149.517
C02975=1131.454,108.224,-56.352,-179.897,8.102,149.517
C02976=1131.449,108.473,-56.371,-179.895,8.107,149.518
C02977=1131.444,108.723,-56.390,-179.893,8.110,149.518
C02978=1131.440,108.971,-56.408,-179.890,8.114,149.518
C02979=1131.435,109.221,-56.428,-179.887,8.119,149.518
C02980=1131.430,109.470,-56.447,-179.885,8.122,149.519
C02981=1131.425,109.720,-56.466,-179.882,8.126,149.519
C02982=1131.420,109.969,-56.485,-179.879,8.130,149.519
C02983=1131.416,110.218,-56.504,-179.877,8.135,149.519
C02984=1131.411,110.467,-56.523,-179.875,8.138,149.519
C02985=1131.407,110.716,-56.542,-179.872,8.142,149.519
C02986=1131.401,110.965,-56.562,-179.869,8.147,149.520
C02987=1131.396,111.215,-56.580,-179.867,8.150,149.520
C02988=1131.392,111.464,-56.599,-179.865,8.154,149.520
C02989=1131.387,111.713,-56.619,-179.863,8.157,149.520
C02990=1131.382,111.962,-56.638,-179.861,8.161,149.521
C02991=1131.377,112.212,-56.658,-179.859,8.164,149.521
C02992=1131.372,112.460,-56.676,-179.857,8.168,149.521
C02993=1131.367,112.710,-56.696,-179.855,8.172,149.521
C02994=1131.363,112.959,-56.716,-179.853,8.175,149.522
C02995=1131.358,113.208,-56.734,-179.851,8.179,149.522
C02996=1131.353,113.457,-56.754,-179.849,8.182,149.522
C02997=1131.348,113.706,-56.773,-179.848,8.186,149.522
C02998=1131.343,113.956,-56.793,-179.845,8.189,149.523
C02999=1131.339,114.204,-56.812,-179.844,8.192,149.523
C03000=1131.334,114.454,-56.831,-179.842,8.196,149.523
C03001=1131.329,114.704,-56.851,-179.840,8.199,149.523
C03002=1131.324,114.952,-56.870,-179.838,8.203,149.524
C03003=1131.319,115.202,-56.890,-179.836,8.206,149.524
C03004=1131.315,115.451,-56.909,-179.834,8.210,149.524
C03005=1131.310,115.700,-56.928,-179.832,8.213,149.524
C03006=1131.305,115.950,-56.948,-179.830,8.217,149.525
C03007=1131.300,116.164,-56.965,-179.829,8.220,149.525
C03008=1131.296,116.379,-56.982,-179.827,8.223,149.525
C03009=1131.293,116.594,-56.999,-179.825,8.226,149.525
C03010=1131.288,116.809,-57.016,-179.824,8.229,149.526
C03011=1131.284,117.024,-57.033,-179.822,8.232,149.526
C03012=1131.280,117.239,-57.050,-179.820,8.235,149.526
C03013=1131.276,117.453,-57.066,-179.819,8.238,149.526
C03014=1131.272,117.668,-57.083,-179.817,8.241,149.526
C03015=1131.268,117.918,-57.102,-179.815,8.245,149.527
C03016=1131.262,118.167,-57.122,-179.813,8.248,149.527
C03017=1131.257,118.416,-57.141,-179.812,8.251,149.527
C03018=1131.253,118.666,-57.161,-179.809,8.255,149.527
C03019=1131.248,118.914,-57.181,-179.807,8.258,149.528
C03020=1131.243,119.164,-57.201,-179.805,8.262,149.528
C03021=1131.238,119.413,-57.220,-179.803,8.265,149.528
C03022=1131.233,119.663,-57.240,-179.802,8.269,149.529
C03023=1131.228,119.911,-57.260,-179.800,8.272,149.529
C03024=1131.224,120.160,-57.279,-179.798,8.275,149.529
C03025=1131.220,120.410,-57.299,-179.796,8.279,149.529
C03026=1131.215,120.658,-57.319,-179.794,8.282,149.529
C03027=1131.210,120.908,-57.338,-179.792,8.286,149.530
C03028=1131.205,121.157,-57.358,-179.791,8.289,149.530
C03029=1131.201,121.406,-57.378,-179.789,8.292,149.530
C03030=1131.195,121.655,-57.398,-179.787,8.296,149.531
C03031=1131.191,121.905,-57.417,-179.785,8.299,149.531
C03032=1131.186,122.154,-57.438,-179.783,8.303,149.531
C03033=1131.181,122.403,-57.457,-179.782,8.306,149.531
C03034=1131.176,122.652,-57.477,-179.780,8.309,149.532
C03035=1131.172,122.901,-57.497,-179.778,8.313,149.532
C03036=1131.167,123.151,-57.517,-179.775,8.316,149.532
C03037=1131.162,123.399,-57.537,-179.774,8.319,149.533
C03038=1131.158,123.649,-57.557,-179.772,8.323,149.533
C03039=1131.152,123.898,-57.577,-179.770,8.326,149.533
C03040=1131.147,124.147,-57.597,-179.768,8.330,149.533
C03041=1131.143,124.396,-57.617,-179.767,8.333,149.533
C03042=1131.138,124.646,-57.637,-179.765,8.337,149.534
C03043=1131.134,124.895,-57.657,-179.763,8.340,149.534
C03044=1131.128,125.144,-57.677,-179.762,8.343,149.534
C03045=1131.124,125.392,-57.697,-179.760,8.346,149.535
C03046=1131.119,125.642,-57.717,-179.758,8.350,149.535
C03047=1131.115,125.891,-57.737,-179.756,8.354,149.535
C03048=1131.110,126.141,-57.757,-179.754,8.356,149.535
C03049=1131.105,126.390,-57.777,-179.752,8.360,149.536
C03050=1131.099,126.639,-57.797,-179.750,8.363,149.536
C03051=1131.095,126.888,-57.817,-179.749,8.366,149.536
C03052=1131.090,127.137,-57.838,-179.747,8.370,149.536
C03053=1131.086,127.386,-57.857,-179.745,8.373,149.537
C03054=1131.081,127.635,-57.878,-179.744,8.376,149.537
C03055=1131.077,127.885,-57.897,-179.742,8.380,149.537
C03056=1131.071,128.134,-57.918,-179.740,8.384,149.538
C03057=1131.067,128.383,-57.939,-179.739,8.386,149.538
C03058=1131.062,128.632,-57.958,-179.737,8.390,149.538
C03059=1131.057,128.881,-57.978,-179.736,8.393,149.538
C03060=1131.053,129.130,-57.999,-179.733,8.396,149.539
C03061=1131.048,129.379,-58.020,-179.731,8.400,149.539
C03062=1131.043,129.628,-58.039,-179.730,8.403,149.539
C03063=1131.039,129.843,-58.057,-179.729,8.406,149.540
C03064=1131.035,130.058,-58.074,-179.727,8.409,149.540
C03065=1131.031,130.273,-58.093,-179.725,8.412,149.540
C03066=1131.026,130.487,-58.109,-179.724,8.415,149.540
C03067=1131.023,130.702,-58.127,-179.723,8.417,149.540
C03068=1131.018,130.917,-58.145,-179.721,8.420,149.541
C03069=1131.014,131.132,-58.163,-179.720,8.423,149.541
C03070=1131.010,131.347,-58.180,-179.719,8.426,149.541
C03071=1131.006,131.596,-58.200,-179.717,8.429,149.542
C03072=1131.001,131.845,-58.221,-179.715,8.432,149.542
C03073=1130.996,132.094,-58.241,-179.714,8.436,149.542
C03074=1130.991,132.344,-58.261,-179.711,8.439,149.542
C03075=1130.986,132.593,-58.282,-179.710,8.442,149.543
C03076=1130.982,132.842,-58.302,-179.708,8.446,149.543
C03077=1130.977,133.090,-58.322,-179.707,8.449,149.543
C03078=1130.972,133.339,-58.343,-179.705,8.452,149.544
C03079=1130.967,133.588,-58.364,-179.704,8.455,149.544
C03080=1130.963,133.837,-58.384,-179.702,8.459,149.544
C03081=1130.957,134.087,-58.404,-179.700,8.461,149.544
C03082=1130.953,134.336,-58.425,-179.699,8.465,149.545
C03083=1130.948,134.585,-58.445,-179.697,8.469,149.545
C03084=1130.943,134.834,-58.466,-179.696,8.472,149.546
C03085=1130.939,135.083,-58.486,-179.694,8.475,149.546
C03086=1130.934,135.332,-58.507,-179.692,8.478,149.546
C03087=1130.929,135.581,-58.528,-179.690,8.482,149.546
C03088=1130.925,135.830,-58.548,-179.689,8.485,149.547
C03089=1130.920,136.080,-58.569,-179.687,8.489,149.547
C03090=1130.915,136.329,-58.589,-179.686,8.491,149.547
C03091=1130.911,136.579,-58.611,-179.684,8.495,149.548
C03092=1130.906,136.827,-58.631,-179.683,8.498,149.548
C03093=1130.901,137.077,-58.652,-179.681,8.501,149.548
C03094=1130.897,137.326,-58.672,-179.680,8.504,149.549
C03095=1130.892,137.575,-58.693,-179.678,8.508,149.549
C03096=1130.887,137.824,-58.714,-179.677,8.511,149.549
C03097=1130.882,138.073,-58.734,-179.675,8.515,149.549
C03098=1130.877,138.322,-58.755,-179.674,8.518,149.550
C03099=1130.873,138.571,-58.776,-179.672,8.521,149.550
C03100=1130.868,138.820,-58.797,-179.671,8.524,149.551
C03101=1130.864,139.069,-58.818,-179.668,8.528,149.551
C03102=1130.858,139.318,-58.839,-179.667,8.531,149.551
C03103=1130.854,139.567,-58.859,-179.665,8.534,149.551
C03104=1130.849,139.816,-58.880,-179.664,8.537,149.552
C03105=1130.844,140.065,-58.900,-179.663,8.540,149.552
C03106=1130.840,140.315,-58.922,-179.661,8.544,149.553
C03107=1130.835,140.564,-58.942,-179.660,8.547,149.553
C03108=1130.830,140.813,-58.964,-179.658,8.551,149.553
C03109=1130.825,141.062,-58.985,-179.657,8.554,149.554
C03110=1130.821,141.311,-59.005,-179.655,8.557,149.554
C03111=1130.816,141.560,-59.026,-179.654,8.560,149.554
C03112=1130.811,141.809,-59.046,-179.652,8.564,149.554
C03113=1130.806,142.058,-59.068,-179.651,8.567,149.555
C03114=1130.803,142.307,-59.089,-179.650,8.570,149.555
C03115=1130.797,142.557,-59.110,-179.648,8.573,149.556
C03116=1130.792,142.806,-59.131,-179.647,8.576,149.556
C03117=1130.788,143.054,-59.152,-179.645,8.580,149.556
C03118=1130.783,143.303,-59.173,-179.644,8.583,149.557
C03119=1130.779,143.518,-59.191,-179.643,8.586,149.557
C03120=1130.775,143.733,-59.209,-179.641,8.589,149.557
C03121=1130.771,143.947,-59.227,-179.640,8.592,149.558
C03122=1130.767,144.162,-59.245,-179.639,8.595,149.558
C03123=1130.762,144.377,-59.263,-179.637,8.597,149.558
C03124=1130.759,144.591,-59.281,-179.636,8.600,149.559
C03125=1130.754,144.806,-59.300,-179.635,8.603,149.559
C03126=1130.751,145.021,-59.317,-179.634,8.606,149.559
C03127=1130.746,145.271,-59.339,-179.632,8.610,149.560
C03128=1130.741,145.519,-59.360,-179.629,8.614,149.560
C03129=1130.736,145.769,-59.381,-179.626,8.618,149.560
C03130=1130.732,146.017,-59.402,-179.623,8.622,149.560
C03131=1130.727,146.266,-59.423,-179.620,8.626,149.560
C03132=1130.722,146.516,-59.445,-179.617,8.630,149.560
C03133=1130.718,146.764,-59.466,-179.615,8.635,149.560
C03134=1130.713,147.014,-59.487,-179.612,8.638,149.561
C03135=1130.708,147.262,-59.508,-179.609,8.642,149.561
C03136=1130.703,147.512,-59.530,-179.607,8.646,149.561
C03137=1130.699,147.761,-59.551,-179.604,8.650,149.561
C03138=1130.694,148.010,-59.572,-179.601,8.654,149.561
C03139=1130.689,148.259,-59.594,-179.598,8.657,149.561
C03140=1130.685,148.508,-59.615,-179.596,8.662,149.562
C03141=1130.680,148.757,-59.637,-179.593,8.666,149.562
C03142=1130.676,149.005,-59.658,-179.590,8.669,149.562
C03143=1130.671,149.255,-59.679,-179.588,8.673,149.562
C03144=1130.666,149.504,-59.701,-179.585,8.677,149.562
C03145=1130.661,149.753,-59.722,-179.582,8.681,149.562
C03146=1130.656,150.002,-59.743,-179.579,8.685,149.562
C03147=1130.652,150.251,-59.765,-179.577,8.689,149.563
C03148=1130.647,150.501,-59.786,-179.573,8.693,149.563
C03149=1130.643,150.749,-59.807,-179.571,8.696,149.563
C03150=1130.638,150.998,-59.829,-179.568,8.700,149.563
C03151=1130.633,151.247,-59.850,-179.566,8.704,149.563
C03152=1130.628,151.496,-59.872,-179.563,8.707,149.563
C03153=1130.624,151.745,-59.894,-179.560,8.712,149.563
C03154=1130.619,151.994,-59.916,-179.558,8.715,149.563
C03155=1130.614,152.243,-59.937,-179.555,8.719,149.564
C03156=1130.610,152.493,-59.959,-179.553,8.722,149.564
C03157=1130.605,152.741,-59.981,-179.550,8.726,149.564
C03158=1130.600,152.990,-60.002,-179.547,8.730,149.564
C03159=1130.596,153.239,-60.024,-179.545,8.734,149.564
C03160=1130.591,153.488,-60.046,-179.542,8.737,149.564
C03161=1130.586,153.738,-60.067,-179.539,8.741,149.564
C03162=1130.581,153.987,-60.089,-179.537,8.744,149.564
C03163=1130.577,154.235,-60.111,-179.534,8.748,149.564
C03164=1130.572,154.485,-60.133,-179.532,8.752,149.565
C03165=1130.567,154.733,-60.154,-179.528,8.756,149.565
C03166=1130.563,154.983,-60.176,-179.526,8.759,149.565
C03167=1130.558,155.231,-60.198,-179.523,8.763,149.565
C03168=1130.554,155.481,-60.220,-179.521,8.766,149.565
C03169=1130.549,155.729,-60.242,-179.519,8.770,149.565
C03170=1130.545,155.978,-60.264,-179.515,8.773,149.565
C03171=1130.539,156.227,-60.286,-179.513,8.777,149.565
C03172=1130.534,156.476,-60.308,-179.510,8.781,149.566
C03173=1130.530,156.725,-60.330,-179.508,8.784,149.566
C03174=1130.525,156.974,-60.352,-179.505,8.787,149.566
C03175=1130.522,157.189,-60.371,-179.503,8.791,149.566
C03176=1130.517,157.404,-60.389,-179.501,8.794,149.566
C03177=1130.513,157.618,-60.408,-179.498,8.797,149.566
C03178=1130.510,157.833,-60.428,-179.496,8.799,149.566
C03179=1130.505,158.048,-60.446,-179.494,8.803,149.566
C03180=1130.501,158.262,-60.465,-179.492,8.806,149.566
C03181=1130.497,158.476,-60.484,-179.490,8.808,149.566
C03182=1130.493,158.692,-60.503,-179.488,8.811,149.566
C03183=1130.489,158.940,-60.526,-179.485,8.815,149.566
C03184=1130.484,159.189,-60.548,-179.482,8.818,149.566
C03185=1130.479,159.438,-60.570,-179.479,8.822,149.566
C03186=1130.475,159.687,-60.592,-179.477,8.825,149.567
C03187=1130.471,159.937,-60.614,-179.475,8.828,149.567
C03188=1130.466,160.185,-60.636,-179.472,8.832,149.567
C03189=1130.461,160.434,-60.659,-179.469,8.836,149.567
C03190=1130.456,160.683,-60.681,-179.467,8.839,149.567
C03191=1130.452,160.932,-60.703,-179.464,8.842,149.567
C03192=1130.447,161.180,-60.725,-179.462,8.845,149.567
C03193=1130.442,161.430,-60.748,-179.459,8.849,149.567
C03194=1130.438,161.679,-60.770,-179.457,8.852,149.567
C03195=1130.433,161.928,-60.792,-179.454,8.855,149.567
C03196=1130.428,162.177,-60.815,-179.452,8.858,149.567
C03197=1130.424,162.426,-60.837,-179.450,8.862,149.568
C03198=1130.419,162.675,-60.859,-179.447,8.865,149.568
C03199=1130.415,162.924,-60.882,-179.444,8.868,149.568
C03200=1130.410,163.173,-60.904,-179.442,8.871,149.568
C03201=1130.406,163.421,-60.926,-179.439,8.876,149.568
C03202=1130.401,163.671,-60.949,-179.437,8.879,149.568
C03203=1130.396,163.920,-60.971,-179.434,8.882,149.568
C03204=1130.392,164.168,-60.994,-179.432,8.885,149.568
C03205=1130.386,164.417,-61.016,-179.430,8.888,149.568
C03206=1130.382,164.666,-61.039,-179.427,8.891,149.568
C03207=1130.377,164.916,-61.061,-179.425,8.895,149.568
C03208=1130.373,165.164,-61.084,-179.422,8.898,149.568
C03209=1130.368,165.413,-61.106,-179.420,8.901,149.569
C03210=1130.364,165.662,-61.129,-179.417,8.904,149.569
C03211=1130.360,165.911,-61.151,-179.415,8.907,149.569
C03212=1130.354,166.160,-61.174,-179.412,8.910,149.569
C03213=1130.350,166.409,-61.196,-179.410,8.914,149.569
C03214=1130.345,166.658,-61.219,-179.408,8.917,149.569
C03215=1130.340,166.907,-61.241,-179.405,8.920,149.569
C03216=1130.336,167.156,-61.265,-179.403,8.923,149.569
C03217=1130.332,167.404,-61.287,-179.400,8.926,149.569
C03218=1130.326,167.653,-61.310,-179.398,8.930,149.569
C03219=1130.322,167.902,-61.332,-179.396,8.933,149.569
C03220=1130.317,168.151,-61.356,-179.393,8.936,149.569
C03221=1130.313,168.400,-61.378,-179.391,8.938,149.569
C03222=1130.308,168.649,-61.401,-179.389,8.942,149.570
C03223=1130.304,168.898,-61.424,-179.387,8.945,149.570
C03224=1130.299,169.147,-61.446,-179.384,8.948,149.570
C03225=1130.294,169.396,-61.470,-179.381,8.951,149.570
C03226=1130.290,169.644,-61.492,-179.379,8.955,149.570
C03227=1130.285,169.894,-61.515,-179.377,8.958,149.570
C03228=1130.281,170.143,-61.537,-179.374,8.961,149.570
C03229=1130.276,170.392,-61.561,-179.372,8.963,149.570
C03230=1130.271,170.641,-61.584,-179.370,8.967,149.570
C03231=1130.267,170.855,-61.603,-179.368,8.970,149.570
C03232=1130.264,171.070,-61.623,-179.366,8.972,149.570
C03233=1130.259,171.284,-61.642,-179.364,8.974,149.570
C03234=1130.256,171.499,-61.662,-179.362,8.977,149.570
C03235=1130.251,171.713,-61.682,-179.360,8.980,149.571
C03236=1130.247,171.928,-61.702,-179.358,8.983,149.571
C03237=1130.244,172.142,-61.721,-179.356,8.985,149.571
C03238=1130.239,172.357,-61.741,-179.354,8.987,149.571
C03239=1130.235,172.606,-61.765,-179.352,8.991,149.571
C03240=1130.230,172.854,-61.787,-179.350,8.994,149.571
C03241=1130.225,173.103,-61.811,-179.347,8.997,149.571
C03242=1130.221,173.352,-61.834,-179.345,8.999,149.571
C03243=1130.217,173.601,-61.857,-179.343,9.003,149.571
C03244=1130.212,173.850,-61.880,-179.341,9.006,149.571
C03245=1130.207,174.099,-61.903,-179.338,9.009,149.571
C03246=1130.203,174.348,-61.925,-179.336,9.011,149.571
C03247=1130.198,174.596,-61.948,-179.334,9.015,149.572
C03248=1130.193,174.845,-61.972,-179.332,9.018,149.572
C03249=1130.188,175.094,-61.995,-179.329,9.021,149.572
C03250=1130.184,175.343,-62.018,-179.328,9.024,149.572
C03251=1130.180,175.592,-62.041,-179.325,9.027,149.572
C03252=1130.175,175.841,-62.065,-179.323,9.030,149.572
C03253=1130.170,176.090,-62.088,-179.321,9.033,149.572
C03254=1130.166,176.339,-62.111,-179.319,9.036,149.572
C03255=1130.162,176.588,-62.134,-179.316,9.039,149.572
C03256=1130.156,176.836,-62.157,-179.315,9.042,149.573
C03257=1130.152,177.085,-62.181,-179.312,9.045,149.573
C03258=1130.147,177.334,-62.205,-179.310,9.047,149.573
C03259=1130.143,177.583,-62.228,-179.308,9.050,149.573
C03260=1130.139,177.831,-62.251,-179.306,9.054,149.573
C03261=1130.134,178.080,-62.274,-179.304,9.056,149.573
C03262=1130.129,178.330,-62.297,-179.302,9.059,149.573
C03263=1130.125,178.579,-62.321,-179.300,9.062,149.573
C03264=1130.120,178.828,-62.344,-179.297,9.065,149.573
C03265=1130.115,179.077,-62.367,-179.295,9.068,149.574
C03266=1130.111,179.325,-62.391,-179.293,9.071,149.574
C03267=1130.107,179.574,-62.414,-179.290,9.074,149.573
C03268=1130.102,179.823,-62.438,-179.287,9.078,149.573
C03269=1130.097,180.072,-62.461,-179.283,9.082,149.574
C03270=1130.093,180.320,-62.485,-179.280,9.085,149.573
C03271=1130.088,180.569,-62.508,-179.277,9.089,149.573
C03272=1130.084,180.818,-62.532,-179.275,9.092,149.573
C03273=1130.079,181.067,-62.555,-179.271,9.095,149.573
C03274=1130.074,181.316,-62.579,-179.269,9.098,149.573
C03275=1130.070,181.565,-62.603,-179.265,9.102,149.573
C03276=1130.065,181.814,-62.626,-179.262,9.105,149.573
C03277=1130.061,182.062,-62.650,-179.259,9.109,149.573
C03278=1130.056,182.311,-62.673,-179.256,9.111,149.573
C03279=1130.051,182.560,-62.697,-179.254,9.115,149.573
C03280=1130.047,182.809,-62.721,-179.251,9.118,149.573
C03281=1130.042,183.058,-62.744,-179.248,9.122,149.573
C03282=1130.038,183.306,-62.768,-179.245,9.124,149.573
C03283=1130.033,183.555,-62.792,-179.243,9.127,149.573
C03284=1130.028,183.804,-62.815,-179.240,9.131,149.573
C03285=1130.024,184.053,-62.839,-179.237,9.134,149.573
C03286=1130.020,184.302,-62.863,-179.234,9.137,149.573
C03287=1130.015,184.516,-62.883,-179.232,9.139,149.573
C03288=1130.011,184.731,-62.904,-179.230,9.143,149.573
C03289=1130.008,184.945,-62.924,-179.228,9.145,149.573
C03290=1130.004,185.160,-62.945,-179.225,9.148,149.573
C03291=1130.000,185.374,-62.965,-179.223,9.150,149.573
C03292=1129.996,185.588,-62.986,-179.221,9.152,149.573
C03293=1129.992,185.803,-63.007,-179.218,9.155,149.573
C03294=1129.989,186.017,-63.027,-179.217,9.158,149.573
C03295=1129.984,186.266,-63.052,-179.214,9.161,149.573
C03296=1129.979,186.515,-63.075,-179.211,9.164,149.573
C03297=1129.975,186.763,-63.099,-179.209,9.167,149.573
C03298=1129.970,187.012,-63.122,-179.207,9.169,149.573
C03299=1129.966,187.261,-63.146,-179.204,9.172,149.573
C03300=1129.961,187.509,-63.171,-179.202,9.175,149.573
C03301=1129.956,187.759,-63.195,-179.200,9.178,149.573
C03302=1129.952,188.007,-63.219,-179.197,9.181,149.573
C03303=1129.948,188.256,-63.243,-179.195,9.184,149.573
C03304=1129.943,188.505,-63.266,-179.193,9.186,149.573
C03305=1129.938,188.753,-63.290,-179.190,9.189,149.573
C03306=1129.933,189.002,-63.315,-179.188,9.192,149.573
C03307=1129.929,189.252,-63.339,-179.186,9.195,149.573
C03308=1129.925,189.500,-63.363,-179.184,9.197,149.574
C03309=1129.920,189.749,-63.387,-179.181,9.200,149.574
C03310=1129.915,189.998,-63.411,-179.180,9.202,149.574
C03311=1129.911,190.246,-63.435,-179.177,9.206,149.574
C03312=1129.907,190.495,-63.459,-179.176,9.208,149.574
C03313=1129.902,190.744,-63.484,-179.174,9.211,149.574
C03314=1129.897,190.993,-63.508,-179.171,9.214,149.574
C03315=1129.893,191.242,-63.532,-179.169,9.216,149.574
C03316=1129.888,191.490,-63.556,-179.167,9.218,149.574
C03317=1129.884,191.739,-63.581,-179.165,9.222,149.574
C03318=1129.879,191.988,-63.605,-179.163,9.224,149.574
C03319=1129.875,192.236,-63.629,-179.161,9.226,149.574
C03320=1129.870,192.485,-63.653,-179.160,9.229,149.575
C03321=1129.866,192.735,-63.677,-179.158,9.232,149.575
C03322=1129.861,192.983,-63.701,-179.156,9.235,149.575
C03323=1129.856,193.232,-63.726,-179.154,9.237,149.575
C03324=1129.852,193.480,-63.750,-179.152,9.240,149.575
C03325=1129.848,193.729,-63.774,-179.151,9.242,149.575
C03326=1129.843,193.978,-63.799,-179.149,9.245,149.575
C03327=1129.838,194.227,-63.823,-179.147,9.247,149.575
C03328=1129.834,194.476,-63.848,-179.146,9.250,149.576
C03329=1129.829,194.724,-63.872,-179.144,9.252,149.576
C03330=1129.825,194.973,-63.896,-179.143,9.255,149.576
C03331=1129.820,195.222,-63.921,-179.142,9.257,149.576
C03332=1129.816,195.471,-63.945,-179.140,9.259,149.576
C03333=1129.811,195.720,-63.969,-179.138,9.262,149.576
C03334=1129.806,195.968,-63.994,-179.137,9.265,149.577
C03335=1129.803,196.218,-64.018,-179.135,9.267,149.577
C03336=1129.797,196.466,-64.043,-179.132,9.271,149.577
C03337=1129.793,196.715,-64.067,-179.128,9.275,149.577
C03338=1129.789,196.963,-64.092,-179.124,9.279,149.577
C03339=1129.784,197.212,-64.117,-179.120,9.283,149.576
C03340=1129.779,197.461,-64.141,-179.116,9.286,149.576
C03341=1129.775,197.710,-64.166,-179.112,9.290,149.576
C03342=1129.770,197.958,-64.190,-179.108,9.294,149.576
C03343=1129.766,198.173,-64.211,-179.105,9.297,149.576
C03344=1129.763,198.387,-64.233,-179.101,9.300,149.575
C03345=1129.759,198.602,-64.253,-179.098,9.303,149.575
C03346=1129.755,198.816,-64.275,-179.095,9.307,149.575
C03347=1129.752,199.029,-64.296,-179.092,9.310,149.575
C03348=1129.747,199.244,-64.318,-179.089,9.313,149.575
C03349=1129.743,199.458,-64.339,-179.086,9.316,149.575
C03350=1129.739,199.673,-64.360,-179.083,9.319,149.575
C03351=1129.735,199.921,-64.385,-179.079,9.322,149.575
C03352=1129.731,200.170,-64.410,-179.076,9.326,149.575
C03353=1129.726,200.419,-64.434,-179.072,9.329,149.574
C03354=1129.721,200.667,-64.458,-179.068,9.332,149.574
C03355=1129.717,200.916,-64.484,-179.065,9.336,149.574
C03356=1129.712,201.165,-64.509,-179.062,9.339,149.574
C03357=1129.708,201.413,-64.534,-179.058,9.342,149.574
C03358=1129.703,201.662,-64.559,-179.054,9.346,149.573
C03359=1129.699,201.911,-64.584,-179.051,9.348,149.573
C03360=1129.695,202.159,-64.609,-179.048,9.352,149.573
C03361=1129.690,202.409,-64.634,-179.045,9.355,149.573
C03362=1129.685,202.657,-64.659,-179.041,9.358,149.573
C03363=1129.682,202.906,-64.683,-179.039,9.361,149.573
C03364=1129.676,203.155,-64.708,-179.035,9.365,149.573
C03365=1129.672,203.403,-64.734,-179.032,9.367,149.573
C03366=1129.667,203.652,-64.758,-179.029,9.370,149.573
C03367=1129.664,203.901,-64.784,-179.026,9.374,149.572
C03368=1129.658,204.149,-64.808,-179.023,9.376,149.572
C03369=1129.654,204.398,-64.834,-179.020,9.379,149.572
C03370=1129.649,204.646,-64.859,-179.017,9.382,149.572
C03371=1129.645,204.896,-64.884,-179.014,9.385,149.572
C03372=1129.641,205.143,-64.909,-179.011,9.388,149.572
C03373=1129.636,205.393,-64.934,-179.008,9.391,149.572
C03374=1129.632,205.642,-64.960,-179.006,9.394,149.572
C03375=1129.627,205.890,-64.985,-179.003,9.396,149.572
C03376=1129.623,206.139,-65.010,-179.000,9.399,149.571
C03377=1129.618,206.387,-65.036,-178.997,9.402,149.572
C03378=1129.614,206.636,-65.060,-178.995,9.405,149.571
C03379=1129.609,206.885,-65.086,-178.992,9.408,149.571
C03380=1129.605,207.133,-65.111,-178.990,9.410,149.571
C03381=1129.601,207.383,-65.136,-178.987,9.413,149.571
C03382=1129.596,207.631,-65.162,-178.984,9.416,149.571
C03383=1129.591,207.880,-65.188,-178.982,9.418,149.571
C03384=1129.587,208.128,-65.213,-178.980,9.421,149.571
C03385=1129.582,208.377,-65.238,-178.977,9.424,149.571
C03386=1129.578,208.626,-65.264,-178.975,9.426,149.571
C03387=1129.573,208.874,-65.289,-178.972,9.430,149.571
C03388=1129.569,209.123,-65.315,-178.971,9.432,149.571
C03389=1129.564,209.371,-65.339,-178.968,9.434,149.571
C03390=1129.560,209.620,-65.365,-178.966,9.437,149.571
C03391=1129.556,209.869,-65.390,-178.964,9.439,149.571
C03392=1129.551,210.117,-65.416,-178.962,9.442,149.571
C03393=1129.547,210.366,-65.442,-178.959,9.445,149.571
C03394=1129.542,210.615,-65.467,-178.957,9.447,149.571
C03395=1129.538,210.863,-65.492,-178.956,9.449,149.571
C03396=1129.533,211.112,-65.518,-178.954,9.452,149.572
C03397=1129.529,211.361,-65.544,-178.952,9.455,149.572
C03398=1129.524,211.609,-65.569,-178.950,9.457,149.572
C03399=1129.521,211.824,-65.591,-178.948,9.459,149.572
C03400=1129.517,212.038,-65.613,-178.947,9.462,149.572
C03401=1129.513,212.252,-65.636,-178.945,9.464,149.572
C03402=1129.509,212.466,-65.658,-178.944,9.466,149.572
C03403=1129.505,212.680,-65.679,-178.942,9.468,149.572
C03404=1129.501,212.895,-65.702,-178.941,9.470,149.572
C03405=1129.498,213.109,-65.723,-178.940,9.473,149.573
C03406=1129.494,213.323,-65.746,-178.939,9.474,149.573
C03407=1129.489,213.571,-65.772,-178.937,9.477,149.573
C03408=1129.484,213.819,-65.797,-178.935,9.480,149.573
C03409=1129.480,214.068,-65.823,-178.933,9.483,149.573
C03410=1129.476,214.317,-65.849,-178.931,9.485,149.573
C03411=1129.472,214.566,-65.874,-178.929,9.488,149.573
C03412=1129.467,214.814,-65.900,-178.927,9.491,149.574
C03413=1129.463,215.063,-65.925,-178.925,9.493,149.574
C03414=1129.459,215.312,-65.951,-178.924,9.496,149.574
C03415=1129.454,215.561,-65.978,-178.921,9.499,149.574
C03416=1129.449,215.809,-66.003,-178.920,9.502,149.574
C03417=1129.445,216.058,-66.029,-178.917,9.505,149.574
C03418=1129.440,216.306,-66.054,-178.916,9.507,149.574
C03419=1129.436,216.555,-66.080,-178.913,9.511,149.575
C03420=1129.431,216.803,-66.106,-178.912,9.513,149.575
C03421=1129.427,217.052,-66.131,-178.909,9.516,149.575
C03422=1129.423,217.301,-66.157,-178.908,9.519,149.575
C03423=1129.418,217.550,-66.183,-178.905,9.522,149.575
C03424=1129.413,217.798,-66.209,-178.903,9.525,149.575
C03425=1129.409,218.046,-66.235,-178.900,9.528,149.575
C03426=1129.405,218.295,-66.261,-178.899,9.531,149.575
C03427=1129.401,218.544,-66.287,-178.896,9.534,149.576
C03428=1129.396,218.793,-66.313,-178.893,9.537,149.576
C03429=1129.391,219.041,-66.339,-178.891,9.540,149.576
C03430=1129.387,219.289,-66.365,-178.888,9.543,149.576
C03431=1129.383,219.538,-66.391,-178.886,9.547,149.576
C03432=1129.378,219.787,-66.416,-178.884,9.550,149.576
C03433=1129.374,220.035,-66.444,-178.881,9.553,149.576
C03434=1129.370,220.284,-66.469,-178.879,9.556,149.576
C03435=1129.365,220.532,-66.495,-178.876,9.559,149.576
C03436=1129.360,220.781,-66.521,-178.874,9.562,149.576
C03437=1129.356,221.030,-66.547,-178.871,9.566,149.576
C03438=1129.352,221.278,-66.573,-178.869,9.569,149.576
C03439=1129.347,221.527,-66.599,-178.866,9.572,149.576
C03440=1129.343,221.776,-66.626,-178.864,9.575,149.577
C03441=1129.339,222.025,-66.652,-178.861,9.578,149.577
C03442=1129.334,222.273,-66.677,-178.858,9.582,149.577
C03443=1129.329,222.521,-66.704,-178.855,9.585,149.577
C03444=1129.325,222.770,-66.730,-178.852,9.588,149.577
C03445=1129.321,223.018,-66.756,-178.849,9.592,149.577
C03446=1129.316,223.267,-66.783,-178.847,9.595,149.577
C03447=1129.312,223.515,-66.809,-178.844,9.597,149.577
C03448=1129.307,223.765,-66.836,-178.841,9.601,149.577
C03449=1129.303,224.013,-66.861,-178.838,9.604,149.577
C03450=1129.299,224.262,-66.888,-178.834,9.608,149.577
C03451=1129.294,224.511,-66.914,-178.832,9.611,149.577
C03452=1129.289,224.758,-66.940,-178.828,9.615,149.577
C03453=1129.285,225.007,-66.967,-178.826,9.618,149.577
C03454=1129.281,225.255,-66.993,-178.822,9.621,149.577
C03455=1129.277,225.470,-67.016,-178.820,9.624,149.577
C03456=1129.273,225.683,-67.039,-178.817,9.627,149.577
C03457=1129.270,225.898,-67.062,-178.814,9.630,149.577
C03458=1129.265,226.112,-67.084,-178.811,9.633,149.576
C03459=1129.261,226.326,-67.107,-178.809,9.636,149.576
C03460=1129.258,226.540,-67.130,-178.806,9.639,149.576
C03461=1129.254,226.754,-67.153,-178.803,9.642,149.576
C03462=1129.250,226.968,-67.176,-178.800,9.645,149.576
C03463=1129.246,227.216,-67.203,-178.797,9.648,149.576
C03464=1129.241,227.465,-67.229,-178.793,9.652,149.576
C03465=1129.238,227.714,-67.255,-178.790,9.655,149.576
C03466=1129.233,227.962,-67.282,-178.786,9.659,149.576
C03467=1129.229,228.211,-67.308,-178.782,9.662,149.576
C03468=1129.224,228.459,-67.335,-178.779,9.666,149.576
C03469=1129.219,228.708,-67.362,-178.775,9.669,149.575
C03470=1129.215,228.956,-67.389,-178.772,9.673,149.575
C03471=1129.211,229.205,-67.416,-178.768,9.676,149.575
C03472=1129.207,229.453,-67.442,-178.765,9.680,149.575
C03473=1129.202,229.702,-67.469,-178.761,9.683,149.575
C03474=1129.197,229.950,-67.496,-178.757,9.687,149.575
C03475=1129.193,230.199,-67.522,-178.753,9.690,149.575
C03476=1129.189,230.447,-67.549,-178.750,9.694,149.574
C03477=1129.184,230.696,-67.576,-178.746,9.697,149.574
C03478=1129.181,230.944,-67.603,-178.742,9.700,149.574
C03479=1129.176,231.193,-67.630,-178.739,9.703,149.574
C03480=1129.171,231.441,-67.657,-178.736,9.707,149.574
C03481=1129.167,231.690,-67.684,-178.732,9.710,149.574
C03482=1129.163,231.938,-67.711,-178.729,9.713,149.574
C03483=1129.158,232.187,-67.738,-178.725,9.716,149.573
C03484=1129.154,232.435,-67.765,-178.722,9.719,149.573
C03485=1129.149,232.684,-67.792,-178.719,9.722,149.573
C03486=1129.146,232.932,-67.819,-178.715,9.726,149.573
C03487=1129.141,233.181,-67.846,-178.712,9.729,149.573
C03488=1129.136,233.429,-67.873,-178.709,9.731,149.573
C03489=1129.132,233.678,-67.900,-178.706,9.735,149.572
C03490=1129.127,233.926,-67.927,-178.703,9.738,149.572
C03491=1129.123,234.175,-67.954,-178.699,9.740,149.572
C03492=1129.119,234.423,-67.982,-178.696,9.743,149.572
C03493=1129.115,234.672,-68.009,-178.693,9.746,149.572
C03494=1129.110,234.920,-68.036,-178.690,9.749,149.572
C03495=1129.105,235.169,-68.063,-178.687,9.752,149.572
C03496=1129.101,235.417,-68.090,-178.684,9.754,149.571
C03497=1129.098,235.665,-68.117,-178.681,9.757,149.571
C03498=1129.093,235.914,-68.145,-178.678,9.760,149.571
C03499=1129.088,236.162,-68.172,-178.675,9.763,149.571
C03500=1129.084,236.411,-68.199,-178.673,9.766,149.571
C03501=1129.080,236.660,-68.227,-178.670,9.769,149.571
C03502=1129.075,236.908,-68.254,-178.667,9.770,149.571
C03503=1129.071,237.157,-68.281,-178.664,9.773,149.571
C03504=1129.066,237.405,-68.308,-178.661,9.776,149.571
C03505=1129.062,237.654,-68.336,-178.658,9.779,149.570
C03506=1129.058,237.902,-68.363,-178.657,9.781,149.571
C03507=1129.053,238.151,-68.390,-178.654,9.784,149.570
C03508=1129.049,238.399,-68.418,-178.651,9.787,149.570
C03509=1129.044,238.648,-68.445,-178.649,9.789,149.570
C03510=1129.040,238.896,-68.473,-178.646,9.792,149.570
C03511=1129.037,239.110,-68.496,-178.643,9.794,149.570
C03512=1129.033,239.323,-68.520,-178.642,9.796,149.570
C03513=1129.029,239.538,-68.544,-178.639,9.798,149.570
C03514=1129.026,239.751,-68.568,-178.638,9.799,149.570
C03515=1129.021,239.965,-68.591,-178.636,9.801,149.570
C03516=1129.018,240.179,-68.615,-178.634,9.804,149.570
C03517=1129.015,240.393,-68.639,-178.632,9.806,149.570
C03518=1129.010,240.607,-68.662,-178.630,9.808,149.570
C03519=1129.006,240.855,-68.690,-178.628,9.810,149.570
C03520=1129.001,241.104,-68.717,-178.625,9.812,149.570
C03521=1128.997,241.352,-68.745,-178.623,9.815,149.570
C03522=1128.993,241.601,-68.772,-178.622,9.817,149.570
C03523=1128.989,241.849,-68.800,-178.619,9.820,149.570
C03524=1128.985,242.098,-68.828,-178.617,9.822,149.570
C03525=1128.980,242.346,-68.855,-178.615,9.824,149.570
C03526=1128.976,242.594,-68.882,-178.613,9.827,149.570
C03527=1128.972,242.843,-68.911,-178.612,9.828,149.570
C03528=1128.966,243.092,-68.938,-178.610,9.831,149.570
C03529=1128.962,243.340,-68.966,-178.608,9.833,149.570
C03530=1128.958,243.588,-68.994,-178.606,9.835,149.570
C03531=1128.954,243.837,-69.021,-178.604,9.838,149.570
C03532=1128.949,244.084,-69.049,-178.602,9.840,149.570
C03533=1128.946,244.333,-69.077,-178.601,9.842,149.570
C03534=1128.941,244.582,-69.104,-178.599,9.844,149.570
C03535=1128.937,244.830,-69.132,-178.598,9.847,149.571
C03536=1128.932,245.079,-69.160,-178.596,9.848,149.571
C03537=1128.927,245.327,-69.188,-178.594,9.850,149.571
C03538=1128.924,245.575,-69.216,-178.593,9.853,149.571
C03539=1128.919,245.824,-69.243,-178.592,9.855,149.571
C03540=1128.915,246.072,-69.271,-178.590,9.857,149.571
C03541=1128.911,246.320,-69.299,-178.589,9.859,149.571
C03542=1128.905,246.569,-69.327,-178.587,9.862,149.572
C03543=1128.902,246.818,-69.355,-178.586,9.863,149.572
C03544=1128.897,247.066,-69.383,-178.585,9.865,149.572
C03545=1128.894,247.314,-69.411,-178.584,9.868,149.572
C03546=1128.889,247.563,-69.438,-178.579,9.872,149.572
C03547=1128.884,247.811,-69.466,-178.572,9.877,149.571
C03548=1128.880,248.059,-69.494,-178.566,9.882,149.571
C03549=1128.876,248.307,-69.522,-178.559,9.887,149.570
C03550=1128.871,248.556,-69.551,-178.553,9.892,149.570
C03551=1128.867,248.805,-69.578,-178.546,9.898,149.569
C03552=1128.863,249.053,-69.606,-178.540,9.902,149.569
C03553=1128.859,249.301,-69.634,-178.534,9.906,149.568
C03554=1128.854,249.550,-69.662,-178.529,9.910,149.568
C03555=1128.850,249.798,-69.690,-178.524,9.915,149.567
C03556=1128.845,250.047,-69.719,-178.518,9.919,149.567
C03557=1128.841,250.295,-69.747,-178.513,9.922,149.566
C03558=1128.837,250.543,-69.775,-178.509,9.926,149.566
C03559=1128.833,250.792,-69.804,-178.505,9.929,149.566
C03560=1128.828,251.040,-69.831,-178.501,9.932,149.566
C03561=1128.824,251.288,-69.861,-178.497,9.936,149.565
C03562=1128.820,251.536,-69.889,-178.493,9.938,149.565
C03563=1128.815,251.785,-69.917,-178.490,9.941,149.565
C03564=1128.811,252.033,-69.945,-178.487,9.944,149.565
C03565=1128.806,252.282,-69.974,-178.484,9.946,149.564
C03566=1128.803,252.530,-70.002,-178.481,9.948,149.564
C03567=1128.799,252.744,-70.027,-178.479,9.951,149.564
C03568=1128.795,252.958,-70.052,-178.477,9.952,149.564
C03569=1128.792,253.171,-70.075,-178.475,9.954,149.564
C03570=1128.788,253.385,-70.100,-178.474,9.955,149.564
C03571=1128.784,253.599,-70.124,-178.472,9.957,149.564
C03572=1128.780,253.812,-70.149,-178.471,9.959,149.564
C03573=1128.776,254.026,-70.174,-178.471,9.959,149.564
C03574=1128.773,254.240,-70.198,-178.469,9.961,149.564
C03575=1128.769,254.488,-70.227,-178.469,9.962,149.564
C03576=1128.765,254.736,-70.255,-178.468,9.963,149.564
C03577=1128.760,254.985,-70.284,-178.468,9.964,149.565
C03578=1128.756,255.234,-70.312,-178.468,9.965,149.565
C03579=1128.751,255.482,-70.340,-178.468,9.967,149.565
C03580=1128.747,255.730,-70.370,-178.469,9.967,149.566
C03581=1128.743,255.978,-70.397,-178.469,9.968,149.566
C03582=1128.738,256.227,-70.426,-178.467,9.970,149.566
C03583=1128.735,256.475,-70.455,-178.464,9.973,149.566
C03584=1128.730,256.723,-70.483,-178.461,9.976,149.566
C03585=1128.726,256.972,-70.511,-178.458,9.979,149.566
C03586=1128.722,257.221,-70.540,-178.455,9.982,149.565
C03587=1128.717,257.468,-70.569,-178.452,9.985,149.565
C03588=1128.713,257.717,-70.597,-178.449,9.988,149.565
C03589=1128.709,257.966,-70.626,-178.446,9.991,149.565
C03590=1128.704,258.213,-70.655,-178.443,9.994,149.565
C03591=1128.700,258.462,-70.683,-178.440,9.996,149.565
C03592=1128.696,258.710,-70.713,-178.436,10.000,149.565
C03593=1128.691,258.958,-70.741,-178.433,10.003,149.565
C03594=1128.687,259.207,-70.769,-178.430,10.005,149.565
C03595=1128.683,259.455,-70.799,-178.427,10.009,149.565
C03596=1128.679,259.704,-70.827,-178.424,10.012,149.564
C03597=1128.674,259.951,-70.856,-178.420,10.015,149.564
C03598=1128.670,260.200,-70.885,-178.417,10.018,149.564
C03599=1128.666,260.448,-70.914,-178.414,10.020,149.564
C03600=1128.661,260.696,-70.942,-178.410,10.023,149.564
C03601=1128.657,260.945,-70.971,-178.406,10.027,149.564
C03602=1128.653,261.193,-71.000,-178.404,10.030,149.563
C03603=1128.649,261.441,-71.029,-178.400,10.033,149.563
C03604=1128.644,261.689,-71.058,-178.397,10.036,149.563
C03605=1128.640,261.938,-71.087,-178.393,10.039,149.563
C03606=1128.636,262.186,-71.116,-178.389,10.042,149.563
C03607=1128.632,262.435,-71.145,-178.386,10.045,149.562
C03608=1128.628,262.683,-71.174,-178.382,10.048,149.562
C03609=1128.623,262.930,-71.203,-178.378,10.051,149.562
C03610=1128.618,263.179,-71.232,-178.374,10.055,149.562
C03611=1128.614,263.428,-71.261,-178.371,10.057,149.562
C03612=1128.610,263.676,-71.291,-178.367,10.061,149.561
C03613=1128.607,263.924,-71.320,-178.363,10.064,149.561
C03614=1128.602,264.172,-71.348,-178.359,10.067,149.561
C03615=1128.597,264.420,-71.377,-178.355,10.070,149.560
C03616=1128.593,264.669,-71.407,-178.353,10.072,149.560
C03617=1128.589,264.917,-71.436,-178.350,10.075,149.560
C03618=1128.585,265.166,-71.465,-178.348,10.077,149.560
C03619=1128.580,265.414,-71.494,-178.346,10.079,149.560
C03620=1128.576,265.662,-71.524,-178.343,10.082,149.560
C03621=1128.571,265.910,-71.553,-178.341,10.084,149.560
C03622=1128.567,266.158,-71.582,-178.338,10.087,149.560
C03623=1128.564,266.372,-71.608,-178.335,10.089,149.560
C03624=1128.560,266.586,-71.632,-178.333,10.091,149.560
C03625=1128.557,266.800,-71.658,-178.331,10.093,149.560
C03626=1128.553,267.013,-71.683,-178.329,10.095,149.560
C03627=1128.550,267.227,-71.708,-178.326,10.097,149.559
C03628=1128.545,267.440,-71.734,-178.325,10.099,149.559
C03629=1128.542,267.654,-71.759,-178.322,10.101,149.559
C03630=1128.538,267.867,-71.784,-178.320,10.103,149.559
C03631=1128.534,268.115,-71.814,-178.318,10.105,149.559
C03632=1128.530,268.364,-71.843,-178.315,10.108,149.559
C03633=1128.526,268.612,-71.873,-178.312,10.111,149.559
C03634=1128.522,268.860,-71.902,-178.309,10.113,149.559
C03635=1128.517,269.108,-71.931,-178.307,10.115,149.559
C03636=1128.513,269.357,-71.961,-178.304,10.119,149.559
C03637=1128.509,269.605,-71.990,-178.302,10.121,149.559
C03638=1128.505,269.853,-72.020,-178.299,10.123,149.559
C03639=1128.501,270.102,-72.049,-178.296,10.126,149.558
C03640=1128.496,270.349,-72.078,-178.293,10.128,149.558
C03641=1128.492,270.597,-72.108,-178.291,10.131,149.558
C03642=1128.487,270.846,-72.138,-178.288,10.134,149.558
C03643=1128.483,271.094,-72.167,-178.285,10.136,149.558
C03644=1128.478,271.342,-72.197,-178.282,10.139,149.558
C03645=1128.474,271.591,-72.226,-178.278,10.142,149.558
C03646=1128.470,271.839,-72.256,-178.276,10.143,149.557
C03647=1128.466,272.087,-72.286,-178.273,10.146,149.557
C03648=1128.462,272.335,-72.315,-178.270,10.149,149.557
C03649=1128.458,272.583,-72.345,-178.267,10.152,149.557
C03650=1128.454,272.831,-72.374,-178.264,10.155,149.557
C03651=1128.449,273.080,-72.404,-178.261,10.157,149.557
C03652=1128.445,273.328,-72.434,-178.258,10.160,149.557
C03653=1128.441,273.576,-72.464,-178.256,10.163,149.557
C03654=1128.436,273.824,-72.493,-178.252,10.165,149.557
